         $OUT[836] = ($FLAG[330] OR NOT $FLAG[330] AND NOT $FLAG[331] AND NOT $FLAG[332]) AND NOT $FLAG[537]
      ;ENDFOLD
      ;FOLD A860 = (F330 + !F330 & !F331 & !F332) & F537 ;%{SE}%MKUKATPVW %CVW_SPS %VBOASG %P 2:A860 = (F330 + !F330 & !F331 & !F332) & F537, 3: BOASG
         $OUT[860] = ($FLAG[330] OR NOT $FLAG[330] AND NOT $FLAG[331] AND NOT $FLAG[332]) AND $FLAG[537]
      ;ENDFOLD
      ;FOLD Schritt 43 = A4039 ;%{SE}%MKUKATPVW %CVW_SPS %VST_CON %P 2:Schritt 43 = A4039, 3: ST_CON
         IF $OUT[4039] THEN
            PREVSTEP = $APP_INT[5]
            $APP_INT[5] = 43
         ENDIF
      ;ENDFOLD
   ;ENDFOLD
   ;FOLD SCHRITT 43 -- ROB EZ1/SP1/KE1 SZ4 -- ;%{P}%MKUKATPVW,%CSTEP,%VST_NR,%P 1:SCHRITT, 2:43, 3: ROB EZ1/SP1/KE1 SZ4
      ;FOLD ;%{H}
         Case 43
      ;ENDFOLD
      ;FOLD -- RSK Fehlerausgabe KF1/KW1 Initiator/Motor -- ;%{SE}%MKUKATPVW %CVW_COM %VCOMMENT %P 2:-- RSK Fehlerausgabe KF1/KW1 Initiator/Motor --, 3: VW_COMMENT
      ;ENDFOLD
      ;FOLD F322 = !F313 ;%{SE}%MKUKATPVW %CVW_SPS %VBOASG %P 2:F322 = !F313, 3: BOASG
         $FLAG[322] = NOT $FLAG[313]
      ;ENDFOLD
      ;FOLD T7 ( EIN ) = STOP ;%{SE}%MKUKATPVW %CVW_SPS %VTSTOP %P 2:T7 ( EIN ) = STOP, 3: TSTOP
         VW(#SET_TIME,TRUE,7,1,0)
      ;ENDFOLD
      ;FOLD A834 = !F322 & !F537 ;%{SE}%MKUKATPVW %CVW_SPS %VBOASG %P 2:A834 = !F322 & !F537, 3: BOASG
         $OUT[834] = NOT $FLAG[322] AND NOT $FLAG[537]
      ;ENDFOLD
      ;FOLD A858 = !F322 & F537 ;%{SE}%MKUKATPVW %CVW_SPS %VBOASG %P 2:A858 = !F322 & F537, 3: BOASG
         $OUT[858] = NOT $FLAG[322] AND $FLAG[537]
      ;ENDFOLD
      ;FOLD Schritt 44 = !F322 & A4039 ;%{SE}%MKUKATPVW %CVW_SPS %VST_CON %P 2:Schritt 44 = !F322 & A4039, 3: ST_CON
         IF NOT $FLAG[322] AND $OUT[4039] THEN
            PREVSTEP = $APP_INT[5]
            $APP_INT[5] = 44
         ENDIF
      ;ENDFOLD
      ;FOLD Schritt 46 = F322 & A4039 ;%{SE}%MKUKATPVW %CVW_SPS %VST_CON %P 2:Schritt 46 = F322 & A4039, 3: ST_CON
         IF $FLAG[322] AND $OUT[4039] THEN
            PREVSTEP = $APP_INT[5]
            $APP_INT[5] = 46
         ENDIF
      ;ENDFOLD
   ;ENDFOLD
   ;FOLD SCHRITT 44 -- ROB EZ1/SP1/KE1 SZ4 -- ;%{P}%MKUKATPVW,%CSTEP,%VST_NR,%P 1:SCHRITT, 2:44, 3: ROB EZ1/SP1/KE1 SZ4
      ;FOLD ;%{H}
         Case 44
      ;ENDFOLD
      ;FOLD F312 = AUS ;%{SE}%MKUKATPVW %CVW_SPS %VBOASG %P 2:F312 = AUS, 3: BOASG
         $FLAG[312] = FALSE
      ;ENDFOLD
      ;FOLD F313 = AUS ;%{SE}%MKUKATPVW %CVW_SPS %VBOASG %P 2:F313 = AUS, 3: BOASG
         $FLAG[313] = FALSE
      ;ENDFOLD
      ;FOLD -- Umdreh. KF setzen -- ;%{SE}%MKUKATPVW %CVW_COM %VCOMMENT %P 2:-- Umdreh. KF setzen --, 3: VW_COMMENT
      ;ENDFOLD
      ;FOLD i1 ( EIN ) = 0 ;%{SE}%MKUKATPVW %CVW_SPS %VARIASG %P 2:i1 ( EIN ) = 0, 3: ARIASG
         VW(#COUNTER,TRUE,1,0)
      ;ENDFOLD
      ;FOLD -- Ueberwachungszeit EZ1/SP1/KE1 SZ4 schliessen -- ;%{SE}%MKUKATPVW %CVW_COM %VCOMMENT %P 2:-- Ueberwachungszeit EZ1/SP1/KE1 SZ4 schliessen --, 3: VW_COMMENT
      ;ENDFOLD
      ;FOLD T9 ( EIN ) = -40[1/10Sek] ;%{SE}%MKUKATPVW %CVW_SPS %VTASG %P 2:T9 ( EIN ) = -40[1/10Sek], 3: TASG
         VW(#SET_TIME,TRUE,9,0,-40)
      ;ENDFOLD
      ;FOLD -- Ueberwachungszeit KF1 -- ;%{SE}%MKUKATPVW %CVW_COM %VCOMMENT %P 2:-- Ueberwachungszeit KF1 --, 3: VW_COMMENT
      ;ENDFOLD
      ;FOLD T7 ( EIN ) = -40[1/10Sek] ;%{SE}%MKUKATPVW %CVW_SPS %VTASG %P 2:T7 ( EIN ) = -40[1/10Sek], 3: TASG
         VW(#SET_TIME,TRUE,7,0,-40)
      ;ENDFOLD
      ;FOLD Schritt 45 = A4039 ;%{SE}%MKUKATPVW %CVW_SPS %VST_CON %P 2:Schritt 45 = A4039, 3: ST_CON
         IF $OUT[4039] THEN
            PREVSTEP = $APP_INT[5]
            $APP_INT[5] = 45
         ENDIF
      ;ENDFOLD
   ;ENDFOLD
   ;FOLD SCHRITT 45 -- ROB EZ1/SP1/KE1 SZ4 -- ;%{P}%MKUKATPVW,%CSTEP,%VST_NR,%P 1:SCHRITT, 2:45, 3: ROB EZ1/SP1/KE1 SZ4
      ;FOLD ;%{H}
         Case 45
      ;ENDFOLD
      ;FOLD -- KF1/KW1 Ausblasen -- ;%{SE}%MKUKATPVW %CVW_COM %VCOMMENT %P 2:-- KF1/KW1 Ausblasen --, 3: VW_COMMENT
      ;ENDFOLD
      ;FOLD A836 = (F330 + F331 + !F330 & !F331 & !F332) & !F537 ;%{SE}%MKUKATPVW %CVW_SPS %VBOASG %P 2:A836 = (F330 + F331 + !F330 & !F331 & !F332) & !F537, 3: BOASG
         $OUT[836] = ($FLAG[330] OR $FLAG[331] OR NOT $FLAG[330] AND NOT $FLAG[331] AND NOT $FLAG[332]) AND NOT $FLAG[537]
      ;ENDFOLD
      ;FOLD A860 = (F330 + F331 + !F330 & !F331 & !F332) & F537 ;%{SE}%MKUKATPVW %CVW_SPS %VBOASG %P 2:A860 = (F330 + F331 + !F330 & !F331 & !F332) & F537, 3: BOASG
         $OUT[860] = ($FLAG[330] OR $FLAG[331] OR NOT $FLAG[330] AND NOT $FLAG[331] AND NOT $FLAG[332]) AND $FLAG[537]
      ;ENDFOLD
      ;FOLD -- EZ1/SP1/KE1 SZ4 schliessen -- ;%{SE}%MKUKATPVW %CVW_COM %VCOMMENT %P 2:-- EZ1/SP1/KE1 SZ4 schliessen --, 3: VW_COMMENT
      ;ENDFOLD
      ;FOLD A717 = AUS ;%{SE}%MKUKATPVW %CVW_SPS %VBOASG %P 2:A717 = AUS, 3: BOASG
         $OUT[717] = FALSE
      ;ENDFOLD
      ;FOLD -- EZ1/SP1 -- ;%{SE}%MKUKATPVW %CVW_COM %VCOMMENT %P 2:-- EZ1/SP1 --, 3: VW_COMMENT
      ;ENDFOLD
      ;FOLD A718 = !F830 ;%{SE}%MKUKATPVW %CVW_SPS %VBOASG %P 2:A718 = !F830, 3: BOASG
         $OUT[718] = NOT $FLAG[830]
      ;ENDFOLD
      ;FOLD A766 = F830 ;%{SE}%MKUKATPVW %CVW_SPS %VBOASG %P 2:A766 = F830, 3: BOASG
         $OUT[766] = $FLAG[830]
      ;ENDFOLD
      ;FOLD Schritt 46 = (!E717 & E718 + T9) & A4039 ;%{SE}%MKUKATPVW %CVW_SPS %VST_CON %P 2:Schritt 46 = (!E717 & E718 + T9) & A4039, 3: ST_CON
         IF (NOT $IN[717] AND $IN[718] OR $TIMER_FLAG[9]) AND $OUT[4039] THEN
            PREVSTEP = $APP_INT[5]
            $APP_INT[5] = 46
         ENDIF
      ;ENDFOLD
   ;ENDFOLD
   ;FOLD SCHRITT 46 -- ROB EZ1/SP1/KE1 SZ4 -- ;%{P}%MKUKATPVW,%CSTEP,%VST_NR,%P 1:SCHRITT, 2:46, 3: ROB EZ1/SP1/KE1 SZ4
      ;FOLD ;%{H}
         Case 46
      ;ENDFOLD
      ;FOLD T9 ( EIN ) = STOP ;%{SE}%MKUKATPVW %CVW_SPS %VTSTOP %P 2:T9 ( EIN ) = STOP, 3: TSTOP
         VW(#SET_TIME,TRUE,9,1,0)
      ;ENDFOLD
      ;FOLD -- RSK Fehlerausgabe Kraftaufbau -- ;%{SE}%MKUKATPVW %CVW_COM %VCOMMENT %P 2:-- RSK Fehlerausgabe Kraftaufbau --, 3: VW_COMMENT
      ;ENDFOLD
      ;FOLD F325 = T9 ;%{SE}%MKUKATPVW %CVW_SPS %VBOASG %P 2:F325 = T9, 3: BOASG
         $FLAG[325] = $TIMER_FLAG[9]
      ;ENDFOLD
      ;FOLD -- KF1/KW1 abschalten bei Fehler -- ;%{SE}%MKUKATPVW %CVW_COM %VCOMMENT %P 2:-- KF1/KW1 abschalten bei Fehler --, 3: VW_COMMENT
      ;ENDFOLD
      ;FOLD A834 = !T7 & !T9 & !F537 ;%{SE}%MKUKATPVW %CVW_SPS %VBOASG %P 2:A834 = !T7 & !T9 & !F537, 3: BOASG
         $OUT[834] = NOT $TIMER_FLAG[7] AND NOT $TIMER_FLAG[9] AND NOT $FLAG[537]
      ;ENDFOLD
      ;FOLD A858 = !T7 & !T9 & F537 ;%{SE}%MKUKATPVW %CVW_SPS %VBOASG %P 2:A858 = !T7 & !T9 & F537, 3: BOASG
         $OUT[858] = NOT $TIMER_FLAG[7] AND NOT $TIMER_FLAG[9] AND $FLAG[537]
      ;ENDFOLD
      ;FOLD -- KF1/KW1 Ausblasen -- ;%{SE}%MKUKATPVW %CVW_COM %VCOMMENT %P 2:-- KF1/KW1 Ausblasen --, 3: VW_COMMENT
      ;ENDFOLD
      ;FOLD A836 = (F330 + F331 + !F330 & !F331 & !F332) & !T9 & !F537 ;%{SE}%MKUKATPVW %CVW_SPS %VBOASG %P 2:A836 = (F330 + F331 + !F330 & !F331 & !F332) & !T9 & !F537, 3: BOASG
         $OUT[836] = ($FLAG[330] OR $FLAG[331] OR NOT $FLAG[330] AND NOT $FLAG[331] AND NOT $FLAG[332]) AND NOT $TIMER_FLAG[9] AND NOT $FLAG[537]
      ;ENDFOLD
      ;FOLD A860 = (F330 + F331 + !F330 & !F331 & !F332) & !T9 & F537 ;%{SE}%MKUKATPVW %CVW_SPS %VBOASG %P 2:A860 = (F330 + F331 + !F330 & !F331 & !F332) & !T9 & F537, 3: BOASG
         $OUT[860] = ($FLAG[330] OR $FLAG[331] OR NOT $FLAG[330] AND NOT $FLAG[331] AND NOT $FLAG[332]) AND NOT $TIMER_FLAG[9] AND $FLAG[537]
      ;ENDFOLD
      ;FOLD -- Warte Fraesen fertig oder Timeout -- ;%{SE}%MKUKATPVW %CVW_COM %VCOMMENT %P 2:-- Warte Fraesen fertig oder Timeout --, 3: VW_COMMENT
      ;ENDFOLD
      ;FOLD Schritt 47 = (F116 & F79 + F112 & !F287 & F78 + F114 & F287 & F78 + T7 + T9) & A4039 ;%{SE}%MKUKATPVW %CVW_SPS %VST_CON %P 2:Schritt 47 = (F116 & F79 + F112 & !F287 & F78 + F114 & F287 & F78 + T7 + T9) & A4039, 3: ST_CON
         IF ($FLAG[116] AND $FLAG[79] OR $FLAG[112] AND NOT $FLAG[287] AND $FLAG[78] OR $FLAG[114] AND $FLAG[287] AND $FLAG[78] OR $TIMER_FLAG[7] OR $TIMER_FLAG[9]) AND $OUT[4039] THEN
            PREVSTEP = $APP_INT[5]
            $APP_INT[5] = 47
         ENDIF
      ;ENDFOLD
   ;ENDFOLD
   ;FOLD SCHRITT 47 -- ROB EZ1/SP1/KE1 SZ4 -- ;%{P}%MKUKATPVW,%CSTEP,%VST_NR,%P 1:SCHRITT, 2:47, 3: ROB EZ1/SP1/KE1 SZ4
      ;FOLD ;%{H}
         Case 47
      ;ENDFOLD
      ;FOLD -- Hilfsflag SK Programmwechsel -- ;%{SE}%MKUKATPVW %CVW_COM %VCOMMENT %P 2:-- Hilfsflag SK Programmwechsel --, 3: VW_COMMENT
      ;ENDFOLD
      ;FOLD F334 = AUS ;%{SE}%MKUKATPVW %CVW_SPS %VBOASG %P 2:F334 = AUS, 3: BOASG
         $FLAG[334] = FALSE
      ;ENDFOLD
      ;FOLD t7 ( EIN ) = STOP ;%{SE}%MKUKATPVW %CVW_SPS %VTSTOP %P 2:t7 ( EIN ) = STOP, 3: TSTOP
         VW(#SET_TIME,TRUE,7,1,0)
      ;ENDFOLD
      ;FOLD -- KF1/KW1 Ausblasen -- ;%{SE}%MKUKATPVW %CVW_COM %VCOMMENT %P 2:-- KF1/KW1 Ausblasen --, 3: VW_COMMENT
      ;ENDFOLD
      ;FOLD A836 = (F330 + F331 + F332 + !F330 & !F331 & !F332) & !F537 ;%{SE}%MKUKATPVW %CVW_SPS %VBOASG %P 2:A836 = (F330 + F331 + F332 + !F330 & !F331 & !F332) & !F537, 3: BOASG
         $OUT[836] = ($FLAG[330] OR $FLAG[331] OR $FLAG[332] OR NOT $FLAG[330] AND NOT $FLAG[331] AND NOT $FLAG[332]) AND NOT $FLAG[537]
      ;ENDFOLD
      ;FOLD A860 = (F330 + F331 + F332 + !F330 & !F331 & !F332) & F537 ;%{SE}%MKUKATPVW %CVW_SPS %VBOASG %P 2:A860 = (F330 + F331 + F332 + !F330 & !F331 & !F332) & F537, 3: BOASG
         $OUT[860] = ($FLAG[330] OR $FLAG[331] OR $FLAG[332] OR NOT $FLAG[330] AND NOT $FLAG[331] AND NOT $FLAG[332]) AND $FLAG[537]
      ;ENDFOLD
      ;FOLD -- KF Ausblasen Ausschaltverzoegerung starten -- ;%{SE}%MKUKATPVW %CVW_COM %VCOMMENT %P 2:-- KF Ausblasen Ausschaltverzoegerung starten --, 3: VW_COMMENT
      ;ENDFOLD
      ;FOLD F736 = EIN ;%{SE}%MKUKATPVW %CVW_SPS %VBOASG %P 2:F736 = EIN, 3: BOASG
         $FLAG[736] = TRUE
      ;ENDFOLD
      ;FOLD -- EZ1/SP1/KE1 SZ4 oeffnen -- ;%{SE}%MKUKATPVW %CVW_COM %VCOMMENT %P 2:-- EZ1/SP1/KE1 SZ4 oeffnen --, 3: VW_COMMENT
      ;ENDFOLD
      ;FOLD A718 = AUS ;%{SE}%MKUKATPVW %CVW_SPS %VBOASG %P 2:A718 = AUS, 3: BOASG
         $OUT[718] = FALSE
      ;ENDFOLD
      ;FOLD A766 = AUS ;%{SE}%MKUKATPVW %CVW_SPS %VBOASG %P 2:A766 = AUS, 3: BOASG
         $OUT[766] = FALSE
      ;ENDFOLD
      ;FOLD A717 = EIN ;%{SE}%MKUKATPVW %CVW_SPS %VBOASG %P 2:A717 = EIN, 3: BOASG
         $OUT[717] = TRUE
      ;ENDFOLD
      ;FOLD -- RSK Sammelstoerung -- ;%{SE}%MKUKATPVW %CVW_COM %VCOMMENT %P 2:-- RSK Sammelstoerung --, 3: VW_COMMENT
      ;ENDFOLD
      ;FOLD F329 = T7 + T9 ;%{SE}%MKUKATPVW %CVW_SPS %VBOASG %P 2:F329 = T7 + T9, 3: BOASG
         $FLAG[329] = $TIMER_FLAG[7] OR $TIMER_FLAG[9]
      ;ENDFOLD
      ;FOLD -- Hilfsflag Startfraesen -- ;%{SE}%MKUKATPVW %CVW_COM %VCOMMENT %P 2:-- Hilfsflag Startfraesen --, 3: VW_COMMENT
      ;ENDFOLD
      ;FOLD F114 = (F114 & F78 + F116 & F79) & F287 ;%{SE}%MKUKATPVW %CVW_SPS %VBOASG %P 2:F114 = (F114 & F78 + F116 & F79) & F287, 3: BOASG
         $FLAG[114] = ($FLAG[114] AND $FLAG[78] OR $FLAG[116] AND $FLAG[79]) AND $FLAG[287]
      ;ENDFOLD
      ;FOLD F116 = !F130 & F116 + F130 & F287 & F116 ;%{SE}%MKUKATPVW %CVW_SPS %VBOASG %P 2:F116 = !F130 & F116 + F130 & F287 & F116, 3: BOASG
         $FLAG[116] = NOT $FLAG[130] AND $FLAG[116] OR $FLAG[130] AND $FLAG[287] AND $FLAG[116]
      ;ENDFOLD
      ;FOLD F287 = F78 + F79 & F130 ;%{SE}%MKUKATPVW %CVW_SPS %VBOASG %P 2:F287 = F78 + F79 & F130, 3: BOASG
         $FLAG[287] = $FLAG[78] OR $FLAG[79] AND $FLAG[130]
      ;ENDFOLD
      ;FOLD -- Wiederholung beim Startfraesen -- ;%{SE}%MKUKATPVW %CVW_COM %VCOMMENT %P 2:-- Wiederholung beim Startfraesen --, 3: VW_COMMENT
      ;ENDFOLD
      ;FOLD Schritt 44 = E717 & !E718 & (F78 & !F114 + F79 & F130 & !F114) & !F329 & A4039 ;%{SE}%MKUKATPVW %CVW_SPS %VST_CON %P 2:Schritt 44 = E717 & !E718 & (F78 & !F114 + F79 & F130 & !F114) & !F329 & A4039, 3: ST_CON
         IF $IN[717] AND NOT $IN[718] AND ($FLAG[78] AND NOT $FLAG[114] OR $FLAG[79] AND $FLAG[130] AND NOT $FLAG[114]) AND NOT $FLAG[329] AND $OUT[4039] THEN
            PREVSTEP = $APP_INT[5]
            $APP_INT[5] = 44
         ENDIF
      ;ENDFOLD
      ;FOLD -- Weiter wenn Fraesen fertig -- ;%{SE}%MKUKATPVW %CVW_COM %VCOMMENT %P 2:-- Weiter wenn Fraesen fertig --, 3: VW_COMMENT
      ;ENDFOLD
      ;FOLD Schritt 48 = E717 & !E718 & (F79 & F116 & (!F130 + F114) + F78 & F114 + F329) & A4039 ;%{SE}%MKUKATPVW %CVW_SPS %VST_CON %P 2:Schritt 48 = E717 & !E718 & (F79 & F116 & (!F130 + F114) + F78 & F114 + F329) & A4039, 3: ST_CON
         IF $IN[717] AND NOT $IN[718] AND ($FLAG[79] AND $FLAG[116] AND (NOT $FLAG[130] OR $FLAG[114]) OR $FLAG[78] AND $FLAG[114] OR $FLAG[329]) AND $OUT[4039] THEN
            PREVSTEP = $APP_INT[5]
            $APP_INT[5] = 48
         ENDIF
      ;ENDFOLD
      ;FOLD -- Weiter bei Fehler -- ;%{SE}%MKUKATPVW %CVW_COM %VCOMMENT %P 2:-- Weiter bei Fehler --, 3: VW_COMMENT
      ;ENDFOLD
      ;FOLD Schritt 50 = F325 & (E26 + E27) & A4039 ;%{SE}%MKUKATPVW %CVW_SPS %VST_CON %P 2:Schritt 50 = F325 & (E26 + E27) & A4039, 3: ST_CON
         IF $FLAG[325] AND ($IN[26] OR $IN[27]) AND $OUT[4039] THEN
            PREVSTEP = $APP_INT[5]
            $APP_INT[5] = 50
         ENDIF
      ;ENDFOLD
   ;ENDFOLD
   ;FOLD SCHRITT 48 -- ROB EZ1/SP1/KE1 SZ4 -- ;%{P}%MKUKATPVW,%CSTEP,%VST_NR,%P 1:SCHRITT, 2:48, 3: ROB EZ1/SP1/KE1 SZ4
      ;FOLD ;%{H}
         Case 48
      ;ENDFOLD
      ;FOLD A717 = AUS ;%{SE}%MKUKATPVW %CVW_SPS %VBOASG %P 2:A717 = AUS, 3: BOASG
         $OUT[717] = FALSE
      ;ENDFOLD
      ;FOLD -- KF1/KW1 abschalten -- ;%{SE}%MKUKATPVW %CVW_COM %VCOMMENT %P 2:-- KF1/KW1 abschalten --, 3: VW_COMMENT
      ;ENDFOLD
      ;FOLD A834 = AUS ;%{SE}%MKUKATPVW %CVW_SPS %VBOASG %P 2:A834 = AUS, 3: BOASG
         $OUT[834] = FALSE
      ;ENDFOLD
      ;FOLD A858 = AUS ;%{SE}%MKUKATPVW %CVW_SPS %VBOASG %P 2:A858 = AUS, 3: BOASG
         $OUT[858] = FALSE
      ;ENDFOLD
      ;FOLD bin3 ( !F329 ) = 4 ;%{SE}%MKUKATPVW %CVW_SPS %VARIASG %P 2:bin3 ( !F329 ) = 4, 3: ARIASG
         VW(#BINOUT,NOT $FLAG[329],3,4)
      ;ENDFOLD
      ;FOLD -- Wartezeit Programmwechsel SK -- ;%{SE}%MKUKATPVW %CVW_COM %VCOMMENT %P 2:-- Wartezeit Programmwechsel SK --, 3: VW_COMMENT
      ;ENDFOLD
      ;FOLD T8 ( !F334 ) = -2[1/10Sek] ;%{SE}%MKUKATPVW %CVW_SPS %VTASG %P 2:T8 ( !F334 ) = -2[1/10Sek], 3: TASG
         VW(#SET_TIME,NOT $FLAG[334],8,0,-2)
      ;ENDFOLD
      ;FOLD -- Hilfsflag SK Programmwechsel -- ;%{SE}%MKUKATPVW %CVW_COM %VCOMMENT %P 2:-- Hilfsflag SK Programmwechsel --, 3: VW_COMMENT
      ;ENDFOLD
      ;FOLD F334 = EIN ;%{SE}%MKUKATPVW %CVW_SPS %VBOASG %P 2:F334 = EIN, 3: BOASG
         $FLAG[334] = TRUE
      ;ENDFOLD
      ;FOLD Schritt 49 = T8 & A4039 ;%{SE}%MKUKATPVW %CVW_SPS %VST_CON %P 2:Schritt 49 = T8 & A4039, 3: ST_CON
         IF $TIMER_FLAG[8] AND $OUT[4039] THEN
            PREVSTEP = $APP_INT[5]
            $APP_INT[5] = 49
         ENDIF
      ;ENDFOLD
   ;ENDFOLD
   ;FOLD SCHRITT 49 -- ROB EZ1/SP1/KE1 SZ4 -- ;%{P}%MKUKATPVW,%CSTEP,%VST_NR,%P 1:SCHRITT, 2:49, 3: ROB EZ1/SP1/KE1 SZ4
      ;FOLD ;%{H}
         Case 49
      ;ENDFOLD
      ;FOLD -- Hilfsflag SK Programmwechsel -- ;%{SE}%MKUKATPVW %CVW_COM %VCOMMENT %P 2:-- Hilfsflag SK Programmwechsel --, 3: VW_COMMENT
      ;ENDFOLD
      ;FOLD F334 = AUS ;%{SE}%MKUKATPVW %CVW_SPS %VBOASG %P 2:F334 = AUS, 3: BOASG
         $FLAG[334] = FALSE
      ;ENDFOLD
      ;FOLD -- Quitt. Fraesen SK1 -- ;%{SE}%MKUKATPVW %CVW_COM %VCOMMENT %P 2:-- Quitt. Fraesen SK1 --, 3: VW_COMMENT
      ;ENDFOLD
      ;FOLD A786 = !F329 & !F322 ;%{SE}%MKUKATPVW %CVW_SPS %VBOASG %P 2:A786 = !F329 & !F322, 3: BOASG
         $OUT[786] = NOT $FLAG[329] AND NOT $FLAG[322]
      ;ENDFOLD
      ;FOLD Schritt 50 = (!E786 & E787 & !E788 + F329) & A4039 ;%{SE}%MKUKATPVW %CVW_SPS %VST_CON %P 2:Schritt 50 = (!E786 & E787 & !E788 + F329) & A4039, 3: ST_CON
         IF (NOT $IN[786] AND $IN[787] AND NOT $IN[788] OR $FLAG[329]) AND $OUT[4039] THEN
            PREVSTEP = $APP_INT[5]
            $APP_INT[5] = 50
         ENDIF
      ;ENDFOLD
   ;ENDFOLD
   ;FOLD SCHRITT 50 -- ROB EZ1/SP1/KE1 SZ4 # Ende -- ;%{P}%MKUKATPVW,%CSTEP,%VST_NR,%P 1:SCHRITT, 2:50, 3: ROB EZ1/SP1/KE1 SZ4 # Ende
      ;FOLD ;%{H}
         Case 50
      ;ENDFOLD
      ;FOLD -- KF1/KW1 Ausblasen -- ;%{SE}%MKUKATPVW %CVW_COM %VCOMMENT %P 2:-- KF1/KW1 Ausblasen --, 3: VW_COMMENT
      ;ENDFOLD
      ;FOLD A836 = (F330 + F331 + F332) & F736 ;%{SE}%MKUKATPVW %CVW_SPS %VBOASG %P 2:A836 = (F330 + F331 + F332) & F736, 3: BOASG
         $OUT[836] = ($FLAG[330] OR $FLAG[331] OR $FLAG[332]) AND $FLAG[736]
      ;ENDFOLD
      ;FOLD A860 = (F330 + F331 + F332) & F736 ;%{SE}%MKUKATPVW %CVW_SPS %VBOASG %P 2:A860 = (F330 + F331 + F332) & F736, 3: BOASG
         $OUT[860] = ($FLAG[330] OR $FLAG[331] OR $FLAG[332]) AND $FLAG[736]
      ;ENDFOLD
      ;FOLD F91 = !E786 & E787 & !E788 & !F322 & !F325 & !F329 ;%{SE}%MKUKATPVW %CVW_SPS %VBOASG %P 2:F91 = !E786 & E787 & !E788 & !F322 & !F325 & !F329, 3: BOASG
         $FLAG[91] = NOT $IN[786] AND $IN[787] AND NOT $IN[788] AND NOT $FLAG[322] AND NOT $FLAG[325] AND NOT $FLAG[329]
      ;ENDFOLD
      ;FOLD Schritt 39 = (F322 + F325 + F329) & (E26 + E27) & A4039 ;%{SE}%MKUKATPVW %CVW_SPS %VST_CON %P 2:Schritt 39 = (F322 + F325 + F329) & (E26 + E27) & A4039, 3: ST_CON
         IF ($FLAG[322] OR $FLAG[325] OR $FLAG[329]) AND ($IN[26] OR $IN[27]) AND $OUT[4039] THEN
            PREVSTEP = $APP_INT[5]
            $APP_INT[5] = 39
         ENDIF
      ;ENDFOLD
      ;FOLD Schritt 1 = F91 & !F322 & !F325 & !F329 & A4039 ;%{SE}%MKUKATPVW %CVW_SPS %VST_CON %P 2:Schritt 1 = F91 & !F322 & !F325 & !F329 & A4039, 3: ST_CON
         IF $FLAG[91] AND NOT $FLAG[322] AND NOT $FLAG[325] AND NOT $FLAG[329] AND $OUT[4039] THEN
            PREVSTEP = $APP_INT[5]
            $APP_INT[5] = 1
         ENDIF
      ;ENDFOLD
   ;ENDFOLD
   ;FOLD SCHRITT 51 -- STAT EZ1/SP1/KE1 # Start-- ;%{P}%MKUKATPVW,%CSTEP,%VST_NR,%P 1:SCHRITT, 2:51, 3: STAT EZ1/SP1/KE1 # Start
      ;FOLD ;%{H}
         Case 51
      ;ENDFOLD
      ;FOLD -- RSK gestartet -- ;%{SE}%MKUKATPVW %CVW_COM %VCOMMENT %P 2:-- RSK gestartet --, 3: VW_COMMENT
      ;ENDFOLD
      ;FOLD F122 = AUS ;%{SE}%MKUKATPVW %CVW_SPS %VBOASG %P 2:F122 = AUS, 3: BOASG
         $FLAG[122] = FALSE
      ;ENDFOLD
      ;FOLD F321 = AUS ;%{SE}%MKUKATPVW %CVW_SPS %VBOASG %P 2:F321 = AUS, 3: BOASG
         $FLAG[321] = FALSE
      ;ENDFOLD
      ;FOLD F322 = AUS ;%{SE}%MKUKATPVW %CVW_SPS %VBOASG %P 2:F322 = AUS, 3: BOASG
         $FLAG[322] = FALSE
      ;ENDFOLD
      ;FOLD F323 = AUS ;%{SE}%MKUKATPVW %CVW_SPS %VBOASG %P 2:F323 = AUS, 3: BOASG
         $FLAG[323] = FALSE
      ;ENDFOLD
      ;FOLD F324 = AUS ;%{SE}%MKUKATPVW %CVW_SPS %VBOASG %P 2:F324 = AUS, 3: BOASG
         $FLAG[324] = FALSE
      ;ENDFOLD
      ;FOLD F325 = AUS ;%{SE}%MKUKATPVW %CVW_SPS %VBOASG %P 2:F325 = AUS, 3: BOASG
         $FLAG[325] = FALSE
      ;ENDFOLD
      ;FOLD F326 = AUS ;%{SE}%MKUKATPVW %CVW_SPS %VBOASG %P 2:F326 = AUS, 3: BOASG
         $FLAG[326] = FALSE
      ;ENDFOLD
      ;FOLD F327 = AUS ;%{SE}%MKUKATPVW %CVW_SPS %VBOASG %P 2:F327 = AUS, 3: BOASG
         $FLAG[327] = FALSE
      ;ENDFOLD
      ;FOLD F329 = AUS ;%{SE}%MKUKATPVW %CVW_SPS %VBOASG %P 2:F329 = AUS, 3: BOASG
         $FLAG[329] = FALSE
      ;ENDFOLD
      ;FOLD -- EZ1/SP1/KE1 SZ1 Zaehler -- ;%{SE}%MKUKATPVW %CVW_COM %VCOMMENT %P 2:-- EZ1/SP1/KE1 SZ1 Zaehler --, 3: VW_COMMENT
      ;ENDFOLD
      ;FOLD F94 = AUS ;%{SE}%MKUKATPVW %CVW_SPS %VBOASG %P 2:F94 = AUS, 3: BOASG
         $FLAG[94] = FALSE
      ;ENDFOLD
      ;FOLD F95 = AUS ;%{SE}%MKUKATPVW %CVW_SPS %VBOASG %P 2:F95 = AUS, 3: BOASG
         $FLAG[95] = FALSE
      ;ENDFOLD
      ;FOLD F96 = AUS ;%{SE}%MKUKATPVW %CVW_SPS %VBOASG %P 2:F96 = AUS, 3: BOASG
         $FLAG[96] = FALSE
      ;ENDFOLD
      ;FOLD F97 = AUS ;%{SE}%MKUKATPVW %CVW_SPS %VBOASG %P 2:F97 = AUS, 3: BOASG
         $FLAG[97] = FALSE
      ;ENDFOLD
      ;FOLD F98 = AUS ;%{SE}%MKUKATPVW %CVW_SPS %VBOASG %P 2:F98 = AUS, 3: BOASG
         $FLAG[98] = FALSE
      ;ENDFOLD
      ;FOLD F99 = AUS ;%{SE}%MKUKATPVW %CVW_SPS %VBOASG %P 2:F99 = AUS, 3: BOASG
         $FLAG[99] = FALSE
      ;ENDFOLD
      ;FOLD -- Hilfsflags Funktionstest KF Motor -- ;%{SE}%MKUKATPVW %CVW_COM %VCOMMENT %P 2:-- Hilfsflags Funktionstest KF Motor --, 3: VW_COMMENT
      ;ENDFOLD
      ;FOLD F312 = AUS ;%{SE}%MKUKATPVW %CVW_SPS %VBOASG %P 2:F312 = AUS, 3: BOASG
         $FLAG[312] = FALSE
      ;ENDFOLD
      ;FOLD F313 = AUS ;%{SE}%MKUKATPVW %CVW_SPS %VBOASG %P 2:F313 = AUS, 3: BOASG
         $FLAG[313] = FALSE
      ;ENDFOLD
      ;FOLD bin1 ( !F830 ) = 31 ;%{SE}%MKUKATPVW %CVW_SPS %VARIASG %P 2:bin1 ( !F830 ) = 31, 3: ARIASG
         VW(#BINOUT,NOT $FLAG[830],1,31)
      ;ENDFOLD
      ;FOLD bin3 ( EIN ) = 31 ;%{SE}%MKUKATPVW %CVW_SPS %VARIASG %P 2:bin3 ( EIN ) = 31, 3: ARIASG
         VW(#BINOUT,TRUE,3,31)
      ;ENDFOLD
      ;FOLD -- Wartezeit Programmwechsel SK -- ;%{SE}%MKUKATPVW %CVW_COM %VCOMMENT %P 2:-- Wartezeit Programmwechsel SK --, 3: VW_COMMENT
      ;ENDFOLD
      ;FOLD T8 ( !F334 ) = -2[1/10Sek] ;%{SE}%MKUKATPVW %CVW_SPS %VTASG %P 2:T8 ( !F334 ) = -2[1/10Sek], 3: TASG
         VW(#SET_TIME,NOT $FLAG[334],8,0,-2)
      ;ENDFOLD
      ;FOLD -- Hilfsflag SK Programmwechsel -- ;%{SE}%MKUKATPVW %CVW_COM %VCOMMENT %P 2:-- Hilfsflag SK Programmwechsel --, 3: VW_COMMENT
      ;ENDFOLD
      ;FOLD F334 = EIN ;%{SE}%MKUKATPVW %CVW_SPS %VBOASG %P 2:F334 = EIN, 3: BOASG
         $FLAG[334] = TRUE
      ;ENDFOLD
      ;FOLD -- Quitt. Fraesen SK1 AUS -- ;%{SE}%MKUKATPVW %CVW_COM %VCOMMENT %P 2:-- Quitt. Fraesen SK1 AUS --, 3: VW_COMMENT
      ;ENDFOLD
      ;FOLD A786 = AUS ;%{SE}%MKUKATPVW %CVW_SPS %VBOASG %P 2:A786 = AUS, 3: BOASG
         $OUT[786] = FALSE
      ;ENDFOLD
      ;FOLD Schritt 52 = T8 & A4039 ;%{SE}%MKUKATPVW %CVW_SPS %VST_CON %P 2:Schritt 52 = T8 & A4039, 3: ST_CON
         IF $TIMER_FLAG[8] AND $OUT[4039] THEN
            PREVSTEP = $APP_INT[5]
            $APP_INT[5] = 52
         ENDIF
      ;ENDFOLD
   ;ENDFOLD
   ;FOLD SCHRITT 52 -- STAT EZ1/SP1/KE1 -- ;%{P}%MKUKATPVW,%CSTEP,%VST_NR,%P 1:SCHRITT, 2:52, 3: STAT EZ1/SP1/KE1
      ;FOLD ;%{H}
         Case 52
      ;ENDFOLD
      ;FOLD -- Fraeszyklen fuer autom. KF-Umderhung -- ;%{SE}%MKUKATPVW %CVW_COM %VCOMMENT %P 2:-- Fraeszyklen fuer autom. KF-Umderhung --, 3: VW_COMMENT
      ;ENDFOLD
      ;FOLD i36 (EIN) = i36 + 1 ;%{SE}%MKUKATPVW %CVW_SPS %VARIASG %P 2:i36 (EIN) = i36 + 1, 3: ARIASG
         VW(#COUNTER,TRUE,36,$COUNT_I[36] + 1)
      ;ENDFOLD
      ;FOLD -- Hilfsflag SK Programmwechsel -- ;%{SE}%MKUKATPVW %CVW_COM %VCOMMENT %P 2:-- Hilfsflag SK Programmwechsel --, 3: VW_COMMENT
      ;ENDFOLD
      ;FOLD F334 = AUS ;%{SE}%MKUKATPVW %CVW_SPS %VBOASG %P 2:F334 = AUS, 3: BOASG
         $FLAG[334] = FALSE
      ;ENDFOLD
      ;FOLD -- Ueberwachungszeit KF1 EIN -- ;%{SE}%MKUKATPVW %CVW_COM %VCOMMENT %P 2:-- Ueberwachungszeit KF1 EIN --, 3: VW_COMMENT
      ;ENDFOLD
      ;FOLD T7 ( EIN ) = -50[1/10Sek] ;%{SE}%MKUKATPVW %CVW_SPS %VTASG %P 2:T7 ( EIN ) = -50[1/10Sek], 3: TASG
         VW(#SET_TIME,TRUE,7,0,-50)
      ;ENDFOLD
      ;FOLD -- KF1 einschalten -- ;%{SE}%MKUKATPVW %CVW_COM %VCOMMENT %P 2:-- KF1 einschalten --, 3: VW_COMMENT
      ;ENDFOLD
      ;FOLD i1 (EIN) = 0 ;%{SE}%MKUKATPVW %CVW_SPS %VARIASG %P 2:i1 (EIN) = 0, 3: ARIASG
         VW(#COUNTER,TRUE,1,0)
      ;ENDFOLD
      ;FOLD A834 = EIN ;%{SE}%MKUKATPVW %CVW_SPS %VBOASG %P 2:A834 = EIN, 3: BOASG
         $OUT[834] = TRUE
      ;ENDFOLD
      ;FOLD Schritt 53 = A4039 ;%{SE}%MKUKATPVW %CVW_SPS %VST_CON %P 2:Schritt 53 = A4039, 3: ST_CON
         IF $OUT[4039] THEN
            PREVSTEP = $APP_INT[5]
            $APP_INT[5] = 53
         ENDIF
      ;ENDFOLD
   ;ENDFOLD
   ;FOLD SCHRITT 53 -- STAT EZ1/SP1/KE1 -- ;%{P}%MKUKATPVW,%CSTEP,%VST_NR,%P 1:SCHRITT, 2:53, 3: STAT EZ1/SP1/KE1
      ;FOLD ;%{H}
         Case 53
      ;ENDFOLD
      ;FOLD -- Funktionstest KF Motor -- ;%{SE}%MKUKATPVW %CVW_COM %VCOMMENT %P 2:-- Funktionstest KF Motor --, 3: VW_COMMENT
      ;ENDFOLD
      ;FOLD F312 = EIN ;%{SE}%MKUKATPVW %CVW_SPS %VBOASG %P 2:F312 = EIN, 3: BOASG
         $FLAG[312] = TRUE
      ;ENDFOLD
      ;FOLD F313 = i1 > 2 ;%{SE}%MKUKATPVW %CVW_SPS %VBOCMP %P 2:F313 = i1 > 2, 3: BOCMP
         $FLAG[313] = $COUNT_I[1] > 2
      ;ENDFOLD
      ;FOLD Schritt 54 = (F313 + T7) & A4039 ;%{SE}%MKUKATPVW %CVW_SPS %VST_CON %P 2:Schritt 54 = (F313 + T7) & A4039, 3: ST_CON
         IF ($FLAG[313] OR $TIMER_FLAG[7]) AND $OUT[4039] THEN
            PREVSTEP = $APP_INT[5]
            $APP_INT[5] = 54
         ENDIF
      ;ENDFOLD
   ;ENDFOLD
   ;FOLD SCHRITT 54 -- STAT EZ1/SP1/KE1-- ;%{P}%MKUKATPVW,%CSTEP,%VST_NR,%P 1:SCHRITT, 2:54, 3: STAT EZ1/SP1/KE1
      ;FOLD ;%{H}
         Case 54
      ;ENDFOLD
      ;FOLD F312 = AUS ;%{SE}%MKUKATPVW %CVW_SPS %VBOASG %P 2:F312 = AUS, 3: BOASG
         $FLAG[312] = FALSE
      ;ENDFOLD
      ;FOLD -- Ueberwachungszeit KS1 schwenken -- ;%{SE}%MKUKATPVW %CVW_COM %VCOMMENT %P 2:-- Ueberwachungszeit KS1 schwenken --, 3: VW_COMMENT
      ;ENDFOLD
      ;FOLD t8 ( EIN ) = -100[1/10Sek] ;%{SE}%MKUKATPVW %CVW_SPS %VTASG %P 2:t8 ( EIN ) = -100[1/10Sek], 3: TASG
         VW(#SET_TIME,TRUE,8,0,-100)
      ;ENDFOLD
      ;FOLD Schritt 55 = A4039 ;%{SE}%MKUKATPVW %CVW_SPS %VST_CON %P 2:Schritt 55 = A4039, 3: ST_CON
         IF $OUT[4039] THEN
            PREVSTEP = $APP_INT[5]
            $APP_INT[5] = 55
         ENDIF
      ;ENDFOLD
   ;ENDFOLD
   ;FOLD SCHRITT 55 -- STAT EZ1/SP1/KE1 -- ;%{P}%MKUKATPVW,%CSTEP,%VST_NR,%P 1:SCHRITT, 2:55, 3: STAT EZ1/SP1/KE1
      ;FOLD ;%{H}
         Case 55
      ;ENDFOLD
      ;FOLD -- RSK Fehlerausgabe KF1 Initiator/Motor -- ;%{SE}%MKUKATPVW %CVW_COM %VCOMMENT %P 2:-- RSK Fehlerausgabe KF1 Initiator/Motor --, 3: VW_COMMENT
      ;ENDFOLD
      ;FOLD F322 = !F313 ;%{SE}%MKUKATPVW %CVW_SPS %VBOASG %P 2:F322 = !F313, 3: BOASG
         $FLAG[322] = NOT $FLAG[313]
      ;ENDFOLD
      ;FOLD -- RSK Fehlerausgabe KS1 Ruhest. -- ;%{SE}%MKUKATPVW %CVW_COM %VCOMMENT %P 2:-- RSK Fehlerausgabe KS1 Ruhest. --, 3: VW_COMMENT
      ;ENDFOLD
      ;FOLD F323 = (!E836 + E837 + E838 + !E839) & !F324 & !F328 ;%{SE}%MKUKATPVW %CVW_SPS %VBOASG %P 2:F323 = (!E836 + E837 + E838 + !E839) & !F324 & !F328, 3: BOASG
         $FLAG[323] = (NOT $IN[836] OR $IN[837] OR $IN[838] OR NOT $IN[839]) AND NOT $FLAG[324] AND NOT $FLAG[328]
      ;ENDFOLD
      ;FOLD -- RSK Sammelstoerung -- ;%{SE}%MKUKATPVW %CVW_COM %VCOMMENT %P 2:-- RSK Sammelstoerung --, 3: VW_COMMENT
      ;ENDFOLD
      ;FOLD F329 = F322 + F323 + T8 ;%{SE}%MKUKATPVW %CVW_SPS %VBOASG %P 2:F329 = F322 + F323 + T8, 3: BOASG
         $FLAG[329] = $FLAG[322] OR $FLAG[323] OR $TIMER_FLAG[8]
      ;ENDFOLD
      ;FOLD T7 ( EIN ) = STOP ;%{SE}%MKUKATPVW %CVW_SPS %VTSTOP %P 2:T7 ( EIN ) = STOP, 3: TSTOP
         VW(#SET_TIME,TRUE,7,1,0)
      ;ENDFOLD
      ;FOLD A834 = !F322 & !F323 ;%{SE}%MKUKATPVW %CVW_SPS %VBOASG %P 2:A834 = !F322 & !F323, 3: BOASG
         $OUT[834] = NOT $FLAG[322] AND NOT $FLAG[323]
      ;ENDFOLD
      ;FOLD -- KF1 Versetzeinheit vor -- ;%{SE}%MKUKATPVW %CVW_COM %VCOMMENT %P 2:-- KF1 Versetzeinheit vor --, 3: VW_COMMENT
      ;ENDFOLD
      ;FOLD A835 = !F322 & !F323 & F564 ;%{SE}%MKUKATPVW %CVW_SPS %VBOASG %P 2:A835 = !F322 & !F323 & F564, 3: BOASG
         $OUT[835] = NOT $FLAG[322] AND NOT $FLAG[323] AND $FLAG[564]
      ;ENDFOLD
      ;FOLD Schritt 56 = (!F322 & !F323 & (E835 & F564 + !E835 & !F564) + T8) & A4039 ;%{SE}%MKUKATPVW %CVW_SPS %VST_CON %P 2:Schritt 56 = (!F322 & !F323 & (E835 & F564 + !E835 & !F564) + T8) & A4039, 3: ST_CON
         IF (NOT $FLAG[322] AND NOT $FLAG[323] AND ($IN[835] AND $FLAG[564] OR NOT $IN[835] AND NOT $FLAG[564]) OR $TIMER_FLAG[8]) AND $OUT[4039] THEN
            PREVSTEP = $APP_INT[5]
            $APP_INT[5] = 56
         ENDIF
      ;ENDFOLD
      ;FOLD Schritt 72 = (F322 + F323) & !F324 & !F328 & A4039 ;%{SE}%MKUKATPVW %CVW_SPS %VST_CON %P 2:Schritt 72 = (F322 + F323) & !F324 & !F328 & A4039, 3: ST_CON
         IF ($FLAG[322] OR $FLAG[323]) AND NOT $FLAG[324] AND NOT $FLAG[328] AND $OUT[4039] THEN
            PREVSTEP = $APP_INT[5]
            $APP_INT[5] = 72
         ENDIF
      ;ENDFOLD
   ;ENDFOLD
   ;FOLD SCHRITT 56 -- STAT EZ1/SP1/KE1 -- ;%{P}%MKUKATPVW,%CSTEP,%VST_NR,%P 1:SCHRITT, 2:56, 3: STAT EZ1/SP1/KE1
      ;FOLD ;%{H}
         Case 56
      ;ENDFOLD
      ;FOLD -- RSK Sammelstoerung -- ;%{SE}%MKUKATPVW %CVW_COM %VCOMMENT %P 2:-- RSK Sammelstoerung --, 3: VW_COMMENT
      ;ENDFOLD
      ;FOLD F329 = T8 ;%{SE}%MKUKATPVW %CVW_SPS %VBOASG %P 2:F329 = T8, 3: BOASG
         $FLAG[329] = $TIMER_FLAG[8]
      ;ENDFOLD
      ;FOLD F324 = AUS ;%{SE}%MKUKATPVW %CVW_SPS %VBOASG %P 2:F324 = AUS, 3: BOASG
         $FLAG[324] = FALSE
      ;ENDFOLD
      ;FOLD F328 = AUS ;%{SE}%MKUKATPVW %CVW_SPS %VBOASG %P 2:F328 = AUS, 3: BOASG
         $FLAG[328] = FALSE
      ;ENDFOLD
      ;FOLD -- KS1 in Arbeitsstellung schwenken -- ;%{SE}%MKUKATPVW %CVW_COM %VCOMMENT %P 2:-- KS1 in Arbeitsstellung schwenken --, 3: VW_COMMENT
      ;ENDFOLD
      ;FOLD A840 = (F745 + !F714) & E717 & !E837 & (E835 & F564 + !E835 & !F564) ;%{SE}%MKUKATPVW %CVW_SPS %VBOASG %P 2:A840 = (F745 + !F714) & E717 & !E837 & (E835 & F564 + !E835 & !F564), 3: BOASG
         $OUT[840] = ($FLAG[745] OR NOT $FLAG[714]) AND $IN[717] AND NOT $IN[837] AND ($IN[835] AND $FLAG[564] OR NOT $IN[835] AND NOT $FLAG[564])
      ;ENDFOLD
      ;FOLD -- KF1 Ausblasen -- ;%{SE}%MKUKATPVW %CVW_COM %VCOMMENT %P 2:-- KF1 Ausblasen --, 3: VW_COMMENT
      ;ENDFOLD
      ;FOLD A836 = F330 + !F330 & !F331 & !F332 ;%{SE}%MKUKATPVW %CVW_SPS %VBOASG %P 2:A836 = F330 + !F330 & !F331 & !F332, 3: BOASG
         $OUT[836] = $FLAG[330] OR NOT $FLAG[330] AND NOT $FLAG[331] AND NOT $FLAG[332]
      ;ENDFOLD
      ;FOLD Schritt 57 = (F745 + !F714) & E717 & (A840 + E837 + T8) & A4039 ;%{SE}%MKUKATPVW %CVW_SPS %VST_CON %P 2:Schritt 57 = (F745 + !F714) & E717 & (A840 + E837 + T8) & A4039, 3: ST_CON
         IF ($FLAG[745] OR NOT $FLAG[714]) AND $IN[717] AND ($OUT[840] OR $IN[837] OR $TIMER_FLAG[8]) AND $OUT[4039] THEN
            PREVSTEP = $APP_INT[5]
            $APP_INT[5] = 57
         ENDIF
      ;ENDFOLD
   ;ENDFOLD
   ;FOLD SCHRITT 57 -- STAT EZ1/SP1/KE1 -- ;%{P}%MKUKATPVW,%CSTEP,%VST_NR,%P 1:SCHRITT, 2:57, 3: STAT EZ1/SP1/KE1
      ;FOLD ;%{H}
         Case 57
      ;ENDFOLD
      ;FOLD -- RSK Fehlerausgabe KF Versetzeinheit -- ;%{SE}%MKUKATPVW %CVW_COM %VCOMMENT %P 2:-- RSK Fehlerausgabe KF Versetzeinheit --, 3: VW_COMMENT
      ;ENDFOLD
      ;FOLD F328 = !E835 & F564 & !F324 ;%{SE}%MKUKATPVW %CVW_SPS %VBOASG %P 2:F328 = !E835 & F564 & !F324, 3: BOASG
         $FLAG[328] = NOT $IN[835] AND $FLAG[564] AND NOT $FLAG[324]
      ;ENDFOLD
      ;FOLD -- RSK Fehlerausgabe KS1 Arbeitsstellung -- ;%{SE}%MKUKATPVW %CVW_COM %VCOMMENT %P 2:-- RSK Fehlerausgabe KS1 Arbeitsstellung --, 3: VW_COMMENT
      ;ENDFOLD
      ;FOLD F324 = (E836 + !E837 + !E838 + E839) & T8 & (E835 + !F564) + F324 ;%{SE}%MKUKATPVW %CVW_SPS %VBOASG %P 2:F324 = (E836 + !E837 + !E838 + E839) & T8 & (E835 + !F564) + F324, 3: BOASG
         $FLAG[324] = ($IN[836] OR NOT $IN[837] OR NOT $IN[838] OR $IN[839]) AND $TIMER_FLAG[8] AND ($IN[835] OR NOT $FLAG[564]) OR $FLAG[324]
      ;ENDFOLD
      ;FOLD -- RSK Fehlerausgabe EZ/SP min. Oeffnung -- ;%{SE}%MKUKATPVW %CVW_COM %VCOMMENT %P 2:-- RSK Fehlerausgabe EZ/SP min. Oeffnung --, 3: VW_COMMENT
      ;ENDFOLD
      ;FOLD F333 = !F745 ;%{SE}%MKUKATPVW %CVW_SPS %VBOASG %P 2:F333 = !F745, 3: BOASG
         $FLAG[333] = NOT $FLAG[745]
      ;ENDFOLD
      ;FOLD -- RSK Sammelstoerung -- ;%{SE}%MKUKATPVW %CVW_COM %VCOMMENT %P 2:-- RSK Sammelstoerung --, 3: VW_COMMENT
      ;ENDFOLD
      ;FOLD F329 = F324 + F328 + F333 ;%{SE}%MKUKATPVW %CVW_SPS %VBOASG %P 2:F329 = F324 + F328 + F333, 3: BOASG
         $FLAG[329] = $FLAG[324] OR $FLAG[328] OR $FLAG[333]
      ;ENDFOLD
      ;FOLD A834 = !F324 & !F328 ;%{SE}%MKUKATPVW %CVW_SPS %VBOASG %P 2:A834 = !F324 & !F328, 3: BOASG
         $OUT[834] = NOT $FLAG[324] AND NOT $FLAG[328]
      ;ENDFOLD
      ;FOLD -- KF1 Ausblasen -- ;%{SE}%MKUKATPVW %CVW_COM %VCOMMENT %P 2:-- KF1 Ausblasen --, 3: VW_COMMENT
      ;ENDFOLD
      ;FOLD A836 = (F330 + !F330 & !F331 & !F332) & !F324 & !F328 ;%{SE}%MKUKATPVW %CVW_SPS %VBOASG %P 2:A836 = (F330 + !F330 & !F331 & !F332) & !F324 & !F328, 3: BOASG
         $OUT[836] = ($FLAG[330] OR NOT $FLAG[330] AND NOT $FLAG[331] AND NOT $FLAG[332]) AND NOT $FLAG[324] AND NOT $FLAG[328]
      ;ENDFOLD
      ;FOLD A836 = F564 ;%{SE}%MKUKATPVW %CVW_SPS %VBOASG %P 2:A836 = F564, 3: BOASG
         $OUT[836] = $FLAG[564]
      ;ENDFOLD
      ;FOLD -- Ueberwachungszeit EZ1/SP1/KE1 SZ1 schliessen -- ;%{SE}%MKUKATPVW %CVW_COM %VCOMMENT %P 2:-- Ueberwachungszeit EZ1/SP1/KE1 SZ1 schliessen --, 3: VW_COMMENT
      ;ENDFOLD
      ;FOLD t9 ( EIN ) = -80[1/10Sek] ;%{SE}%MKUKATPVW %CVW_SPS %VTASG %P 2:t9 ( EIN ) = -80[1/10Sek], 3: TASG
         VW(#SET_TIME,TRUE,9,0,-80)
      ;ENDFOLD
      ;FOLD -- Verweilzeit Versetzeinheit Rueck -- ;%{SE}%MKUKATPVW %CVW_COM %VCOMMENT %P 2:-- Verweilzeit Versetzeinheit Rueck --, 3: VW_COMMENT
      ;ENDFOLD
      ;FOLD t11 ( EIN ) = i24[1/10Sek] ;%{SE}%MKUKATPVW %CVW_SPS %VTASG %P 2:t11 ( EIN ) = i24[1/10Sek], 3: TASG
         VW(#SET_TIME,TRUE,11,0,$COUNT_I[24])
      ;ENDFOLD
      ;FOLD Schritt 52 = (F324 + F328) & (E26 + E27) & A4039 ;%{SE}%MKUKATPVW %CVW_SPS %VST_CON %P 2:Schritt 52 = (F324 + F328) & (E26 + E27) & A4039, 3: ST_CON
         IF ($FLAG[324] OR $FLAG[328]) AND ($IN[26] OR $IN[27]) AND $OUT[4039] THEN
            PREVSTEP = $APP_INT[5]
            $APP_INT[5] = 52
         ENDIF
      ;ENDFOLD
      ;FOLD Schritt 58 = !F324 & !F328 & !E836 & E837 & E838 & !E839 & A4039 ;%{SE}%MKUKATPVW %CVW_SPS %VST_CON %P 2:Schritt 58 = !F324 & !F328 & !E836 & E837 & E838 & !E839 & A4039, 3: ST_CON
         IF NOT $FLAG[324] AND NOT $FLAG[328] AND NOT $IN[836] AND $IN[837] AND $IN[838] AND NOT $IN[839] AND $OUT[4039] THEN
            PREVSTEP = $APP_INT[5]
            $APP_INT[5] = 58
         ENDIF
      ;ENDFOLD
   ;ENDFOLD
   ;FOLD SCHRITT 58 -- STAT EZ1/SP1/KE1-- ;%{P}%MKUKATPVW,%CSTEP,%VST_NR,%P 1:SCHRITT, 2:58, 3: STAT EZ1/SP1/KE1
      ;FOLD ;%{H}
         Case 58
      ;ENDFOLD
      ;FOLD -- Umdreh. KF setzen zwischenspeichern -- ;%{SE}%MKUKATPVW %CVW_COM %VCOMMENT %P 2:-- Umdreh. KF setzen zwischenspeichern --, 3: VW_COMMENT
      ;ENDFOLD
      ;FOLD i45 ( EIN ) = i4 ;%{SE}%MKUKATPVW %CVW_SPS %VARIASG %P 2:i45 ( EIN ) = i4, 3: ARIASG
         VW(#COUNTER,TRUE,45,$COUNT_I[4])
      ;ENDFOLD
      ;FOLD i4 ( F99 ) = i33 ;%{SE}%MKUKATPVW %CVW_SPS %VARIASG %P 2:i4 ( F99 ) = i33, 3: ARIASG
         VW(#COUNTER,$FLAG[99],4,$COUNT_I[33])
      ;ENDFOLD
      ;FOLD i1 ( EIN ) = 0 ;%{SE}%MKUKATPVW %CVW_SPS %VARIASG %P 2:i1 ( EIN ) = 0, 3: ARIASG
         VW(#COUNTER,TRUE,1,0)
      ;ENDFOLD
      ;FOLD F98 = AUS ;%{SE}%MKUKATPVW %CVW_SPS %VBOASG %P 2:F98 = AUS, 3: BOASG
         $FLAG[98] = FALSE
      ;ENDFOLD
      ;FOLD F312 = AUS ;%{SE}%MKUKATPVW %CVW_SPS %VBOASG %P 2:F312 = AUS, 3: BOASG
         $FLAG[312] = FALSE
      ;ENDFOLD
      ;FOLD F313 = AUS ;%{SE}%MKUKATPVW %CVW_SPS %VBOASG %P 2:F313 = AUS, 3: BOASG
         $FLAG[313] = FALSE
      ;ENDFOLD
      ;FOLD F324 = AUS ;%{SE}%MKUKATPVW %CVW_SPS %VBOASG %P 2:F324 = AUS, 3: BOASG
         $FLAG[324] = FALSE
      ;ENDFOLD
      ;FOLD F328 = AUS ;%{SE}%MKUKATPVW %CVW_SPS %VBOASG %P 2:F328 = AUS, 3: BOASG
         $FLAG[328] = FALSE
      ;ENDFOLD
      ;FOLD -- KF1 einschalten nach Fehler -- ;%{SE}%MKUKATPVW %CVW_COM %VCOMMENT %P 2:-- KF1 einschalten nach Fehler --, 3: VW_COMMENT
      ;ENDFOLD
      ;FOLD A834 = EIN ;%{SE}%MKUKATPVW %CVW_SPS %VBOASG %P 2:A834 = EIN, 3: BOASG
         $OUT[834] = TRUE
      ;ENDFOLD
      ;FOLD -- KF1 Versetzeinheit rueck -- ;%{SE}%MKUKATPVW %CVW_COM %VCOMMENT %P 2:-- KF1 Versetzeinheit rueck --, 3: VW_COMMENT
      ;ENDFOLD
      ;FOLD A835 = AUS ;%{SE}%MKUKATPVW %CVW_SPS %VBOASG %P 2:A835 = AUS, 3: BOASG
         $OUT[835] = FALSE
      ;ENDFOLD
      ;FOLD Schritt 59 = T11 & A4039 ;%{SE}%MKUKATPVW %CVW_SPS %VST_CON %P 2:Schritt 59 = T11 & A4039, 3: ST_CON
         IF $TIMER_FLAG[11] AND $OUT[4039] THEN
            PREVSTEP = $APP_INT[5]
            $APP_INT[5] = 59
         ENDIF
      ;ENDFOLD
   ;ENDFOLD
   ;FOLD SCHRITT 59 -- STAT EZ1/SP1/KE1 -- ;%{P}%MKUKATPVW,%CSTEP,%VST_NR,%P 1:SCHRITT, 2:59, 3: STAT EZ1/SP1/KE1
      ;FOLD ;%{H}
         Case 59
      ;ENDFOLD
      ;FOLD t11 ( EIN ) = STOP ;%{SE}%MKUKATPVW %CVW_SPS %VTSTOP %P 2:t11 ( EIN ) = STOP, 3: TSTOP
         VW(#SET_TIME,TRUE,11,1,0)
      ;ENDFOLD
      ;FOLD -- EZ1/SP1/KE1 SZ1 schliessen -- ;%{SE}%MKUKATPVW %CVW_COM %VCOMMENT %P 2:-- EZ1/SP1/KE1 SZ1 schliessen --, 3: VW_COMMENT
      ;ENDFOLD
      ;FOLD A717 = AUS ;%{SE}%MKUKATPVW %CVW_SPS %VBOASG %P 2:A717 = AUS, 3: BOASG
         $OUT[717] = FALSE
      ;ENDFOLD
      ;FOLD -- EZ1/SP1 -- ;%{SE}%MKUKATPVW %CVW_COM %VCOMMENT %P 2:-- EZ1/SP1 --, 3: VW_COMMENT
      ;ENDFOLD
      ;FOLD A718 = !F830 ;%{SE}%MKUKATPVW %CVW_SPS %VBOASG %P 2:A718 = !F830, 3: BOASG
         $OUT[718] = NOT $FLAG[830]
      ;ENDFOLD
      ;FOLD A766 = F830 ;%{SE}%MKUKATPVW %CVW_SPS %VBOASG %P 2:A766 = F830, 3: BOASG
         $OUT[766] = $FLAG[830]
      ;ENDFOLD
      ;FOLD -- KF1 Ausblasen -- ;%{SE}%MKUKATPVW %CVW_COM %VCOMMENT %P 2:-- KF1 Ausblasen --, 3: VW_COMMENT
      ;ENDFOLD
      ;FOLD A836 = F330 + F331 + !F330 & !F331 & !F332 ;%{SE}%MKUKATPVW %CVW_SPS %VBOASG %P 2:A836 = F330 + F331 + !F330 & !F331 & !F332, 3: BOASG
         $OUT[836] = $FLAG[330] OR $FLAG[331] OR NOT $FLAG[330] AND NOT $FLAG[331] AND NOT $FLAG[332]
      ;ENDFOLD
      ;FOLD Schritt 60 = (!E717 & E718 + T9) & A4039 ;%{SE}%MKUKATPVW %CVW_SPS %VST_CON %P 2:Schritt 60 = (!E717 & E718 + T9) & A4039, 3: ST_CON
         IF (NOT $IN[717] AND $IN[718] OR $TIMER_FLAG[9]) AND $OUT[4039] THEN
            PREVSTEP = $APP_INT[5]
            $APP_INT[5] = 60
         ENDIF
      ;ENDFOLD
   ;ENDFOLD
   ;FOLD SCHRITT 60 -- STAT EZ1/SP1/KE1 -- ;%{P}%MKUKATPVW,%CSTEP,%VST_NR,%P 1:SCHRITT, 2:60, 3: STAT EZ1/SP1/KE1
      ;FOLD ;%{H}
         Case 60
      ;ENDFOLD
      ;FOLD -- RSK Fehlerausgabe Kraftaufbau -- ;%{SE}%MKUKATPVW %CVW_COM %VCOMMENT %P 2:-- RSK Fehlerausgabe Kraftaufbau --, 3: VW_COMMENT
      ;ENDFOLD
      ;FOLD F325 = T9 ;%{SE}%MKUKATPVW %CVW_SPS %VBOASG %P 2:F325 = T9, 3: BOASG
         $FLAG[325] = $TIMER_FLAG[9]
      ;ENDFOLD
      ;FOLD -- RSK Sammelstoerung -- ;%{SE}%MKUKATPVW %CVW_COM %VCOMMENT %P 2:-- RSK Sammelstoerung --, 3: VW_COMMENT
      ;ENDFOLD
      ;FOLD F329 = F325 ;%{SE}%MKUKATPVW %CVW_SPS %VBOASG %P 2:F329 = F325, 3: BOASG
         $FLAG[329] = $FLAG[325]
      ;ENDFOLD
      ;FOLD -- KF1 abschalten bei Fehler -- ;%{SE}%MKUKATPVW %CVW_COM %VCOMMENT %P 2:-- KF1 abschalten bei Fehler --, 3: VW_COMMENT
      ;ENDFOLD
      ;FOLD A834 = !T9 ;%{SE}%MKUKATPVW %CVW_SPS %VBOASG %P 2:A834 = !T9, 3: BOASG
         $OUT[834] = NOT $TIMER_FLAG[9]
      ;ENDFOLD
      ;FOLD -- KF1 Ausblasen -- ;%{SE}%MKUKATPVW %CVW_COM %VCOMMENT %P 2:-- KF1 Ausblasen --, 3: VW_COMMENT
      ;ENDFOLD
      ;FOLD A836 = (F330 + F331 + !F330 & !F331 & !F332) & !T9 ;%{SE}%MKUKATPVW %CVW_SPS %VBOASG %P 2:A836 = (F330 + F331 + !F330 & !F331 & !F332) & !T9, 3: BOASG
         $OUT[836] = ($FLAG[330] OR $FLAG[331] OR NOT $FLAG[330] AND NOT $FLAG[331] AND NOT $FLAG[332]) AND NOT $TIMER_FLAG[9]
      ;ENDFOLD
      ;FOLD -- Warte Fraesen fertig oder Timeout -- ;%{SE}%MKUKATPVW %CVW_COM %VCOMMENT %P 2:-- Warte Fraesen fertig oder Timeout --, 3: VW_COMMENT
      ;ENDFOLD
      ;FOLD Schritt 61 = (F79 & F98 + F78 & F94 & !F287 + T7 + T9 + F325) & A4039 ;%{SE}%MKUKATPVW %CVW_SPS %VST_CON %P 2:Schritt 61 = (F79 & F98 + F78 & F94 & !F287 + T7 + T9 + F325) & A4039, 3: ST_CON
         IF ($FLAG[79] AND $FLAG[98] OR $FLAG[78] AND $FLAG[94] AND NOT $FLAG[287] OR $TIMER_FLAG[7] OR $TIMER_FLAG[9] OR $FLAG[325]) AND $OUT[4039] THEN
            PREVSTEP = $APP_INT[5]
            $APP_INT[5] = 61
         ENDIF
      ;ENDFOLD
      ;FOLD Schritt 61 = (F78 & F96 & F287 + T7 + T9 + F325) & A4039 ;%{SE}%MKUKATPVW %CVW_SPS %VST_CON %P 2:Schritt 61 = (F78 & F96 & F287 + T7 + T9 + F325) & A4039, 3: ST_CON
         IF ($FLAG[78] AND $FLAG[96] AND $FLAG[287] OR $TIMER_FLAG[7] OR $TIMER_FLAG[9] OR $FLAG[325]) AND $OUT[4039] THEN
            PREVSTEP = $APP_INT[5]
            $APP_INT[5] = 61
         ENDIF
      ;ENDFOLD
   ;ENDFOLD
   ;FOLD SCHRITT 61 -- STAT EZ1/SP1/KE1-- ;%{P}%MKUKATPVW,%CSTEP,%VST_NR,%P 1:SCHRITT, 2:61, 3: STAT EZ1/SP1/KE1
      ;FOLD ;%{H}
         Case 61
      ;ENDFOLD
      ;FOLD -- EZ1/SP1/KE1 SZ1 oeffnen -- ;%{SE}%MKUKATPVW %CVW_COM %VCOMMENT %P 2:-- EZ1/SP1/KE1 SZ1 oeffnen --, 3: VW_COMMENT
      ;ENDFOLD
      ;FOLD t9 ( EIN ) = STOP ;%{SE}%MKUKATPVW %CVW_SPS %VTSTOP %P 2:t9 ( EIN ) = STOP, 3: TSTOP
         VW(#SET_TIME,TRUE,9,1,0)
      ;ENDFOLD
      ;FOLD A718 = AUS ;%{SE}%MKUKATPVW %CVW_SPS %VBOASG %P 2:A718 = AUS, 3: BOASG
         $OUT[718] = FALSE
      ;ENDFOLD
      ;FOLD A766 = AUS ;%{SE}%MKUKATPVW %CVW_SPS %VBOASG %P 2:A766 = AUS, 3: BOASG
         $OUT[766] = FALSE
      ;ENDFOLD
      ;FOLD A717 = EIN ;%{SE}%MKUKATPVW %CVW_SPS %VBOASG %P 2:A717 = EIN, 3: BOASG
         $OUT[717] = TRUE
      ;ENDFOLD
      ;FOLD -- KF1 Ausblasen -- ;%{SE}%MKUKATPVW %CVW_COM %VCOMMENT %P 2:-- KF1 Ausblasen --, 3: VW_COMMENT
      ;ENDFOLD
      ;FOLD A836 = (F330 + F331 + F332 + !F330 & !F331 & !F332) & !T9 ;%{SE}%MKUKATPVW %CVW_SPS %VBOASG %P 2:A836 = (F330 + F331 + F332 + !F330 & !F331 & !F332) & !T9, 3: BOASG
         $OUT[836] = ($FLAG[330] OR $FLAG[331] OR $FLAG[332] OR NOT $FLAG[330] AND NOT $FLAG[331] AND NOT $FLAG[332]) AND NOT $TIMER_FLAG[9]
      ;ENDFOLD
      ;FOLD -- KF Ausblasen Ausschaltverzoegerung starten -- ;%{SE}%MKUKATPVW %CVW_COM %VCOMMENT %P 2:-- KF Ausblasen Ausschaltverzoegerung starten --, 3: VW_COMMENT
      ;ENDFOLD
      ;FOLD F737 = EIN ;%{SE}%MKUKATPVW %CVW_SPS %VBOASG %P 2:F737 = EIN, 3: BOASG
         $FLAG[737] = TRUE
      ;ENDFOLD
      ;FOLD -- RSK Sammelstoerung -- ;%{SE}%MKUKATPVW %CVW_COM %VCOMMENT %P 2:-- RSK Sammelstoerung --, 3: VW_COMMENT
      ;ENDFOLD
      ;FOLD F329 = T7 + T9 + F325 ;%{SE}%MKUKATPVW %CVW_SPS %VBOASG %P 2:F329 = T7 + T9 + F325, 3: BOASG
         $FLAG[329] = $TIMER_FLAG[7] OR $TIMER_FLAG[9] OR $FLAG[325]
      ;ENDFOLD
      ;FOLD -- Hilfsflag Startfraesen -- ;%{SE}%MKUKATPVW %CVW_COM %VCOMMENT %P 2:-- Hilfsflag Startfraesen --, 3: VW_COMMENT
      ;ENDFOLD
      ;FOLD F96 = F96 & F287 ;%{SE}%MKUKATPVW %CVW_SPS %VBOASG %P 2:F96 = F96 & F287, 3: BOASG
         $FLAG[96] = $FLAG[96] AND $FLAG[287]
      ;ENDFOLD
      ;FOLD F96 = (F96 & F78 + F98 & F79) & F287 ;%{SE}%MKUKATPVW %CVW_SPS %VBOASG %P 2:F96 = (F96 & F78 + F98 & F79) & F287, 3: BOASG
         $FLAG[96] = ($FLAG[96] AND $FLAG[78] OR $FLAG[98] AND $FLAG[79]) AND $FLAG[287]
      ;ENDFOLD
      ;FOLD F98 = !F130 & F98 + F130 & F287 & F98 ;%{SE}%MKUKATPVW %CVW_SPS %VBOASG %P 2:F98 = !F130 & F98 + F130 & F287 & F98, 3: BOASG
         $FLAG[98] = NOT $FLAG[130] AND $FLAG[98] OR $FLAG[130] AND $FLAG[287] AND $FLAG[98]
      ;ENDFOLD
      ;FOLD F287 = F78 + F79 & F130 ;%{SE}%MKUKATPVW %CVW_SPS %VBOASG %P 2:F287 = F78 + F79 & F130, 3: BOASG
         $FLAG[287] = $FLAG[78] OR $FLAG[79] AND $FLAG[130]
      ;ENDFOLD
      ;FOLD -- Neues Fraesprogramm und Zaehler ruecksetzen -- ;%{SE}%MKUKATPVW %CVW_COM %VCOMMENT %P 2:-- Neues Fraesprogramm und Zaehler ruecksetzen --, 3: VW_COMMENT
      ;ENDFOLD
      ;FOLD bin3 ( F130 ) = 36 ;%{SE}%MKUKATPVW %CVW_SPS %VARIASG %P 2:bin3 ( F130 ) = 36, 3: ARIASG
         VW(#BINOUT,$FLAG[130],3,36)
      ;ENDFOLD
      ;FOLD i4 ( F96 ) = i45 ;%{SE}%MKUKATPVW %CVW_SPS %VARIASG %P 2:i4 ( F96 ) = i45, 3: ARIASG
         VW(#COUNTER,$FLAG[96],4,$COUNT_I[45])
      ;ENDFOLD
      ;FOLD -- Wiederholung beim Startfraesen -- ;%{SE}%MKUKATPVW %CVW_COM %VCOMMENT %P 2:-- Wiederholung beim Startfraesen --, 3: VW_COMMENT
      ;ENDFOLD
      ;FOLD Schritt 58 = E717 & !E718 & (F78 & !F96 + F79 & F130 & !F96) & !F329 & A4039 ;%{SE}%MKUKATPVW %CVW_SPS %VST_CON %P 2:Schritt 58 = E717 & !E718 & (F78 & !F96 + F79 & F130 & !F96) & !F329 & A4039, 3: ST_CON
         IF $IN[717] AND NOT $IN[718] AND ($FLAG[78] AND NOT $FLAG[96] OR $FLAG[79] AND $FLAG[130] AND NOT $FLAG[96]) AND NOT $FLAG[329] AND $OUT[4039] THEN
            PREVSTEP = $APP_INT[5]
            $APP_INT[5] = 58
         ENDIF
      ;ENDFOLD
      ;FOLD -- Weiter wenn Fraesen fertig -- ;%{SE}%MKUKATPVW %CVW_COM %VCOMMENT %P 2:-- Weiter wenn Fraesen fertig --, 3: VW_COMMENT
      ;ENDFOLD
      ;FOLD Schritt 62 = E717 & !E718 & (F79 & F98 & (!F130 + F96) + F78 & F96 + F329 + F325) & A4039 ;%{SE}%MKUKATPVW %CVW_SPS %VST_CON %P 2:Schritt 62 = E717 & !E718 & (F79 & F98 & (!F130 + F96) + F78 & F96 + F329 + F325) & A4039, 3: ST_CON
         IF $IN[717] AND NOT $IN[718] AND ($FLAG[79] AND $FLAG[98] AND (NOT $FLAG[130] OR $FLAG[96]) OR $FLAG[78] AND $FLAG[96] OR $FLAG[329] OR $FLAG[325]) AND $OUT[4039] THEN
            PREVSTEP = $APP_INT[5]
            $APP_INT[5] = 62
         ENDIF
      ;ENDFOLD
   ;ENDFOLD
   ;FOLD SCHRITT 62 -- STAT EZ1/SP1/KE1-- ;%{P}%MKUKATPVW,%CSTEP,%VST_NR,%P 1:SCHRITT, 2:62, 3: STAT EZ1/SP1/KE1
      ;FOLD ;%{H}
         Case 62
      ;ENDFOLD
      ;FOLD F324 = AUS ;%{SE}%MKUKATPVW %CVW_SPS %VBOASG %P 2:F324 = AUS, 3: BOASG
         $FLAG[324] = FALSE
      ;ENDFOLD
      ;FOLD A717 = AUS ;%{SE}%MKUKATPVW %CVW_SPS %VBOASG %P 2:A717 = AUS, 3: BOASG
         $OUT[717] = FALSE
      ;ENDFOLD
      ;FOLD -- KF1 abschalten -- ;%{SE}%MKUKATPVW %CVW_COM %VCOMMENT %P 2:-- KF1 abschalten --, 3: VW_COMMENT
      ;ENDFOLD
      ;FOLD A834 = AUS ;%{SE}%MKUKATPVW %CVW_SPS %VBOASG %P 2:A834 = AUS, 3: BOASG
         $OUT[834] = FALSE
      ;ENDFOLD
      ;FOLD -- Ueberwachungszeit KF1 Versetzeinheit -- ;%{SE}%MKUKATPVW %CVW_COM %VCOMMENT %P 2:-- Ueberwachungszeit KF1 Versetzeinheit --, 3: VW_COMMENT
      ;ENDFOLD
      ;FOLD t8 ( EIN ) = -40[1/10Sek] ;%{SE}%MKUKATPVW %CVW_SPS %VTASG %P 2:t8 ( EIN ) = -40[1/10Sek], 3: TASG
         VW(#SET_TIME,TRUE,8,0,-40)
      ;ENDFOLD
      ;FOLD Schritt 63 = A4039 ;%{SE}%MKUKATPVW %CVW_SPS %VST_CON %P 2:Schritt 63 = A4039, 3: ST_CON
         IF $OUT[4039] THEN
            PREVSTEP = $APP_INT[5]
            $APP_INT[5] = 63
         ENDIF
      ;ENDFOLD
   ;ENDFOLD
   ;FOLD SCHRITT 63 -- STAT EZ1/SP1/KE1 -- ;%{P}%MKUKATPVW,%CSTEP,%VST_NR,%P 1:SCHRITT, 2:63, 3: STAT EZ1/SP1/KE1
      ;FOLD ;%{H}
         Case 63
      ;ENDFOLD
      ;FOLD F328 = AUS ;%{SE}%MKUKATPVW %CVW_SPS %VBOASG %P 2:F328 = AUS, 3: BOASG
         $FLAG[328] = FALSE
      ;ENDFOLD
      ;FOLD -- KF1 Versetzeinheit vor -- ;%{SE}%MKUKATPVW %CVW_COM %VCOMMENT %P 2:-- KF1 Versetzeinheit vor --, 3: VW_COMMENT
      ;ENDFOLD
      ;FOLD A835 = F564 ;%{SE}%MKUKATPVW %CVW_SPS %VBOASG %P 2:A835 = F564, 3: BOASG
         $OUT[835] = $FLAG[564]
      ;ENDFOLD
      ;FOLD -- RSK Fehlerausgabe KS1 Arbeitsst. -- ;%{SE}%MKUKATPVW %CVW_COM %VCOMMENT %P 2:-- RSK Fehlerausgabe KS1 Arbeitsst. --, 3: VW_COMMENT
      ;ENDFOLD
      ;FOLD F324 = (E836 + !E837 + !E838 + E839) & !F323 & !F328 + F324 ;%{SE}%MKUKATPVW %CVW_SPS %VBOASG %P 2:F324 = (E836 + !E837 + !E838 + E839) & !F323 & !F328 + F324, 3: BOASG
         $FLAG[324] = ($IN[836] OR NOT $IN[837] OR NOT $IN[838] OR $IN[839]) AND NOT $FLAG[323] AND NOT $FLAG[328] OR $FLAG[324]
      ;ENDFOLD
      ;FOLD -- RSK Sammelstoerung -- ;%{SE}%MKUKATPVW %CVW_COM %VCOMMENT %P 2:-- RSK Sammelstoerung --, 3: VW_COMMENT
      ;ENDFOLD
      ;FOLD F329 = F324 + F325 ;%{SE}%MKUKATPVW %CVW_SPS %VBOASG %P 2:F329 = F324 + F325, 3: BOASG
         $FLAG[329] = $FLAG[324] OR $FLAG[325]
      ;ENDFOLD
      ;FOLD -- Ueberwachungszeit KS1 schwenken -- ;%{SE}%MKUKATPVW %CVW_COM %VCOMMENT %P 2:-- Ueberwachungszeit KS1 schwenken --, 3: VW_COMMENT
      ;ENDFOLD
      ;FOLD t9 ( EIN ) = -100[1/10Sek] ;%{SE}%MKUKATPVW %CVW_SPS %VTASG %P 2:t9 ( EIN ) = -100[1/10Sek], 3: TASG
         VW(#SET_TIME,TRUE,9,0,-100)
      ;ENDFOLD
      ;FOLD Schritt 62 = F324 & (E26 + E27) & A4039 ;%{SE}%MKUKATPVW %CVW_SPS %VST_CON %P 2:Schritt 62 = F324 & (E26 + E27) & A4039, 3: ST_CON
         IF $FLAG[324] AND ($IN[26] OR $IN[27]) AND $OUT[4039] THEN
            PREVSTEP = $APP_INT[5]
            $APP_INT[5] = 62
         ENDIF
      ;ENDFOLD
      ;FOLD Schritt 64 = (!F324 & (E835 & F564 + !E835 & !F564) + T8 + F325) & A4039 ;%{SE}%MKUKATPVW %CVW_SPS %VST_CON %P 2:Schritt 64 = (!F324 & (E835 & F564 + !E835 & !F564) + T8 + F325) & A4039, 3: ST_CON
         IF (NOT $FLAG[324] AND ($IN[835] AND $FLAG[564] OR NOT $IN[835] AND NOT $FLAG[564]) OR $TIMER_FLAG[8] OR $FLAG[325]) AND $OUT[4039] THEN
            PREVSTEP = $APP_INT[5]
            $APP_INT[5] = 64
         ENDIF
      ;ENDFOLD
   ;ENDFOLD
   ;FOLD SCHRITT 64 -- STAT EZ1/SP1/KE1-- ;%{P}%MKUKATPVW,%CSTEP,%VST_NR,%P 1:SCHRITT, 2:64, 3: STAT EZ1/SP1/KE1
      ;FOLD ;%{H}
         Case 64
      ;ENDFOLD
      ;FOLD F323 = AUS ;%{SE}%MKUKATPVW %CVW_SPS %VBOASG %P 2:F323 = AUS, 3: BOASG
         $FLAG[323] = FALSE
      ;ENDFOLD
      ;FOLD F328 = AUS ;%{SE}%MKUKATPVW %CVW_SPS %VBOASG %P 2:F328 = AUS, 3: BOASG
         $FLAG[328] = FALSE
      ;ENDFOLD
      ;FOLD -- RSK Sammelstoerung -- ;%{SE}%MKUKATPVW %CVW_COM %VCOMMENT %P 2:-- RSK Sammelstoerung --, 3: VW_COMMENT
      ;ENDFOLD
      ;FOLD F329 = F325 ;%{SE}%MKUKATPVW %CVW_SPS %VBOASG %P 2:F329 = F325, 3: BOASG
         $FLAG[329] = $FLAG[325]
      ;ENDFOLD
      ;FOLD -- KF1 ein -- ;%{SE}%MKUKATPVW %CVW_COM %VCOMMENT %P 2:-- KF1 ein --, 3: VW_COMMENT
      ;ENDFOLD
      ;FOLD A834 = EIN ;%{SE}%MKUKATPVW %CVW_SPS %VBOASG %P 2:A834 = EIN, 3: BOASG
         $OUT[834] = TRUE
      ;ENDFOLD
      ;FOLD -- KS1 in Ruhestellung schwenken -- ;%{SE}%MKUKATPVW %CVW_COM %VCOMMENT %P 2:-- KS1 in Ruhestellung schwenken --, 3: VW_COMMENT
      ;ENDFOLD
      ;FOLD A840 = (F745 + !F714) & E717 & (E835 & F564 + !E835 & !F564) ;%{SE}%MKUKATPVW %CVW_SPS %VBOASG %P 2:A840 = (F745 + !F714) & E717 & (E835 & F564 + !E835 & !F564), 3: BOASG
         $OUT[840] = ($FLAG[745] OR NOT $FLAG[714]) AND $IN[717] AND ($IN[835] AND $FLAG[564] OR NOT $IN[835] AND NOT $FLAG[564])
      ;ENDFOLD
      ;FOLD Schritt 65 = (F745 + !F714 + T9) & (A840 + T9) & E717 & A4039 ;%{SE}%MKUKATPVW %CVW_SPS %VST_CON %P 2:Schritt 65 = (F745 + !F714 + T9) & (A840 + T9) & E717 & A4039, 3: ST_CON
         IF ($FLAG[745] OR NOT $FLAG[714] OR $TIMER_FLAG[9]) AND ($OUT[840] OR $TIMER_FLAG[9]) AND $IN[717] AND $OUT[4039] THEN
            PREVSTEP = $APP_INT[5]
            $APP_INT[5] = 65
         ENDIF
      ;ENDFOLD
   ;ENDFOLD
   ;FOLD SCHRITT 65 -- STAT EZ1/SP1/KE1 -- ;%{P}%MKUKATPVW,%CSTEP,%VST_NR,%P 1:SCHRITT, 2:65, 3: STAT EZ1/SP1/KE1
      ;FOLD ;%{H}
         Case 65
      ;ENDFOLD
      ;FOLD -- Hilfsflag SK Programmwechsel -- ;%{SE}%MKUKATPVW %CVW_COM %VCOMMENT %P 2:-- Hilfsflag SK Programmwechsel --, 3: VW_COMMENT
      ;ENDFOLD
      ;FOLD F334 = AUS ;%{SE}%MKUKATPVW %CVW_SPS %VBOASG %P 2:F334 = AUS, 3: BOASG
         $FLAG[334] = FALSE
      ;ENDFOLD
      ;FOLD -- RSK Fehlerausgabe KF Versetzeinheit -- ;%{SE}%MKUKATPVW %CVW_COM %VCOMMENT %P 2:-- RSK Fehlerausgabe KF Versetzeinheit --, 3: VW_COMMENT
      ;ENDFOLD
      ;FOLD F328 = !E835 & F564 & !F323 + F328 ;%{SE}%MKUKATPVW %CVW_SPS %VBOASG %P 2:F328 = !E835 & F564 & !F323 + F328, 3: BOASG
         $FLAG[328] = NOT $IN[835] AND $FLAG[564] AND NOT $FLAG[323] OR $FLAG[328]
      ;ENDFOLD
      ;FOLD -- RSK Fehlerausgabe KS1 Ruhestellung -- ;%{SE}%MKUKATPVW %CVW_COM %VCOMMENT %P 2:-- RSK Fehlerausgabe KS1 Ruhestellung --, 3: VW_COMMENT
      ;ENDFOLD
      ;FOLD F323 = (!E836 + E837 + E838 + !E839) & T9 & (E835 + !F564) + F323 ;%{SE}%MKUKATPVW %CVW_SPS %VBOASG %P 2:F323 = (!E836 + E837 + E838 + !E839) & T9 & (E835 + !F564) + F323, 3: BOASG
         $FLAG[323] = (NOT $IN[836] OR $IN[837] OR $IN[838] OR NOT $IN[839]) AND $TIMER_FLAG[9] AND ($IN[835] OR NOT $FLAG[564]) OR $FLAG[323]
      ;ENDFOLD
      ;FOLD -- RSK Fehlerausgabe EZ/SP min. Oeffnung -- ;%{SE}%MKUKATPVW %CVW_COM %VCOMMENT %P 2:-- RSK Fehlerausgabe EZ/SP min. Oeffnung --, 3: VW_COMMENT
      ;ENDFOLD
      ;FOLD F333 = !F745 ;%{SE}%MKUKATPVW %CVW_SPS %VBOASG %P 2:F333 = !F745, 3: BOASG
         $FLAG[333] = NOT $FLAG[745]
      ;ENDFOLD
      ;FOLD -- RSK Sammelstoerung -- ;%{SE}%MKUKATPVW %CVW_COM %VCOMMENT %P 2:-- RSK Sammelstoerung --, 3: VW_COMMENT
      ;ENDFOLD
      ;FOLD F329 = F323 + F325 + F328 + F333 ;%{SE}%MKUKATPVW %CVW_SPS %VBOASG %P 2:F329 = F323 + F325 + F328 + F333, 3: BOASG
         $FLAG[329] = $FLAG[323] OR $FLAG[325] OR $FLAG[328] OR $FLAG[333]
      ;ENDFOLD
      ;FOLD A834 = !F323 & !F328 ;%{SE}%MKUKATPVW %CVW_SPS %VBOASG %P 2:A834 = !F323 & !F328, 3: BOASG
         $OUT[834] = NOT $FLAG[323] AND NOT $FLAG[328]
      ;ENDFOLD
      ;FOLD A836 = F564 ;%{SE}%MKUKATPVW %CVW_SPS %VBOASG %P 2:A836 = F564, 3: BOASG
         $OUT[836] = $FLAG[564]
      ;ENDFOLD
      ;FOLD Schritt 63 = (F323 + F328) & (E26 + E27) & A4039 ;%{SE}%MKUKATPVW %CVW_SPS %VST_CON %P 2:Schritt 63 = (F323 + F328) & (E26 + E27) & A4039, 3: ST_CON
         IF ($FLAG[323] OR $FLAG[328]) AND ($IN[26] OR $IN[27]) AND $OUT[4039] THEN
            PREVSTEP = $APP_INT[5]
            $APP_INT[5] = 63
         ENDIF
      ;ENDFOLD
      ;FOLD Schritt 66 = !A840 & E836 & !E837 & !E838 & E839 & A4039 ;%{SE}%MKUKATPVW %CVW_SPS %VST_CON %P 2:Schritt 66 = !A840 & E836 & !E837 & !E838 & E839 & A4039, 3: ST_CON
         IF NOT $OUT[840] AND $IN[836] AND NOT $IN[837] AND NOT $IN[838] AND $IN[839] AND $OUT[4039] THEN
            PREVSTEP = $APP_INT[5]
            $APP_INT[5] = 66
         ENDIF
      ;ENDFOLD
   ;ENDFOLD
   ;FOLD SCHRITT 66 -- STAT EZ1/SP1/KE1 -- ;%{P}%MKUKATPVW,%CSTEP,%VST_NR,%P 1:SCHRITT, 2:66, 3: STAT EZ1/SP1/KE1
      ;FOLD ;%{H}
         Case 66
      ;ENDFOLD
      ;FOLD F323 = AUS ;%{SE}%MKUKATPVW %CVW_SPS %VBOASG %P 2:F323 = AUS, 3: BOASG
         $FLAG[323] = FALSE
      ;ENDFOLD
      ;FOLD F328 = AUS ;%{SE}%MKUKATPVW %CVW_SPS %VBOASG %P 2:F328 = AUS, 3: BOASG
         $FLAG[328] = FALSE
      ;ENDFOLD
      ;FOLD -- RSK Sammelstoerung -- ;%{SE}%MKUKATPVW %CVW_COM %VCOMMENT %P 2:-- RSK Sammelstoerung --, 3: VW_COMMENT
      ;ENDFOLD
      ;FOLD F329 = F325 ;%{SE}%MKUKATPVW %CVW_SPS %VBOASG %P 2:F329 = F325, 3: BOASG
         $FLAG[329] = $FLAG[325]
      ;ENDFOLD
      ;FOLD t9 ( EIN ) = STOP ;%{SE}%MKUKATPVW %CVW_SPS %VTSTOP %P 2:t9 ( EIN ) = STOP, 3: TSTOP
         VW(#SET_TIME,TRUE,9,1,0)
      ;ENDFOLD
      ;FOLD -- KF1 Versetzeinheit rueck -- ;%{SE}%MKUKATPVW %CVW_COM %VCOMMENT %P 2:-- KF1 Versetzeinheit rueck --, 3: VW_COMMENT
      ;ENDFOLD
      ;FOLD A835 = AUS ;%{SE}%MKUKATPVW %CVW_SPS %VBOASG %P 2:A835 = AUS, 3: BOASG
         $OUT[835] = FALSE
      ;ENDFOLD
      ;FOLD -- KF1 aus -- ;%{SE}%MKUKATPVW %CVW_COM %VCOMMENT %P 2:-- KF1 aus --, 3: VW_COMMENT
      ;ENDFOLD
      ;FOLD A834 = AUS ;%{SE}%MKUKATPVW %CVW_SPS %VBOASG %P 2:A834 = AUS, 3: BOASG
         $OUT[834] = FALSE
      ;ENDFOLD
      ;FOLD -- KF1 Ausblasen -- ;%{SE}%MKUKATPVW %CVW_COM %VCOMMENT %P 2:-- KF1 Ausblasen --, 3: VW_COMMENT
      ;ENDFOLD
      ;FOLD A836 = (F330 + F331 + F332) & F737 ;%{SE}%MKUKATPVW %CVW_SPS %VBOASG %P 2:A836 = (F330 + F331 + F332) & F737, 3: BOASG
         $OUT[836] = ($FLAG[330] OR $FLAG[331] OR $FLAG[332]) AND $FLAG[737]
      ;ENDFOLD
      ;FOLD F168 = !F329 & !F830 ;%{SE}%MKUKATPVW %CVW_SPS %VBOASG %P 2:F168 = !F329 & !F830, 3: BOASG
         $FLAG[168] = NOT $FLAG[329] AND NOT $FLAG[830]
      ;ENDFOLD
      ;FOLD bin1 ( F168 ) = 1 ;%{SE}%MKUKATPVW %CVW_SPS %VARIASG %P 2:bin1 ( F168 ) = 1, 3: ARIASG
         VW(#BINOUT,$FLAG[168],1,1)
      ;ENDFOLD
      ;FOLD F168 = AUS ;%{SE}%MKUKATPVW %CVW_SPS %VBOASG %P 2:F168 = AUS, 3: BOASG
         $FLAG[168] = FALSE
      ;ENDFOLD
      ;FOLD bin3 ( !F329 ) = 1 ;%{SE}%MKUKATPVW %CVW_SPS %VARIASG %P 2:bin3 ( !F329 ) = 1, 3: ARIASG
         VW(#BINOUT,NOT $FLAG[329],3,1)
      ;ENDFOLD
      ;FOLD -- Wartezeit Programmwechsel SK -- ;%{SE}%MKUKATPVW %CVW_COM %VCOMMENT %P 2:-- Wartezeit Programmwechsel SK --, 3: VW_COMMENT
      ;ENDFOLD
      ;FOLD T8 ( !F334 ) = -2[1/10Sek] ;%{SE}%MKUKATPVW %CVW_SPS %VTASG %P 2:T8 ( !F334 ) = -2[1/10Sek], 3: TASG
         VW(#SET_TIME,NOT $FLAG[334],8,0,-2)
      ;ENDFOLD
      ;FOLD -- Hilfsflag SK Programmwechsel -- ;%{SE}%MKUKATPVW %CVW_COM %VCOMMENT %P 2:-- Hilfsflag SK Programmwechsel --, 3: VW_COMMENT
      ;ENDFOLD
      ;FOLD F334 = EIN ;%{SE}%MKUKATPVW %CVW_SPS %VBOASG %P 2:F334 = EIN, 3: BOASG
         $FLAG[334] = TRUE
      ;ENDFOLD
      ;FOLD -- Ueberwachungszeit EZ1/SP1/KE1 SZ1 Messen -- ;%{SE}%MKUKATPVW %CVW_COM %VCOMMENT %P 2:-- Ueberwachungszeit EZ1/SP1/KE1 SZ1 Messen --, 3: VW_COMMENT
      ;ENDFOLD
      ;FOLD t9 ( EIN ) = -150[1/10Sek] ;%{SE}%MKUKATPVW %CVW_SPS %VTASG %P 2:t9 ( EIN ) = -150[1/10Sek], 3: TASG
         VW(#SET_TIME,TRUE,9,0,-150)
      ;ENDFOLD
      ;FOLD Schritt 51 = (F325 + F329) & (E26 + E27) & A4039 ;%{SE}%MKUKATPVW %CVW_SPS %VST_CON %P 2:Schritt 51 = (F325 + F329) & (E26 + E27) & A4039, 3: ST_CON
         IF ($FLAG[325] OR $FLAG[329]) AND ($IN[26] OR $IN[27]) AND $OUT[4039] THEN
            PREVSTEP = $APP_INT[5]
            $APP_INT[5] = 51
         ENDIF
      ;ENDFOLD
      ;FOLD Schritt 67 = T8 & !F325 & !F329 & A4039 ;%{SE}%MKUKATPVW %CVW_SPS %VST_CON %P 2:Schritt 67 = T8 & !F325 & !F329 & A4039, 3: ST_CON
         IF $TIMER_FLAG[8] AND NOT $FLAG[325] AND NOT $FLAG[329] AND $OUT[4039] THEN
            PREVSTEP = $APP_INT[5]
            $APP_INT[5] = 67
         ENDIF
      ;ENDFOLD
   ;ENDFOLD
   ;FOLD SCHRITT 67 -- STAT EZ1/SP1/KE1 -- ;%{P}%MKUKATPVW,%CSTEP,%VST_NR,%P 1:SCHRITT, 2:67, 3: STAT EZ1/SP1/KE1
      ;FOLD ;%{H}
         Case 67
      ;ENDFOLD
      ;FOLD -- Hilfsflag SK Programmwechsel -- ;%{SE}%MKUKATPVW %CVW_COM %VCOMMENT %P 2:-- Hilfsflag SK Programmwechsel --, 3: VW_COMMENT
      ;ENDFOLD
      ;FOLD F334 = AUS ;%{SE}%MKUKATPVW %CVW_SPS %VBOASG %P 2:F334 = AUS, 3: BOASG
         $FLAG[334] = FALSE
      ;ENDFOLD
      ;FOLD -- Quitt. Fraesen SK1 -- ;%{SE}%MKUKATPVW %CVW_COM %VCOMMENT %P 2:-- Quitt. Fraesen SK1 --, 3: VW_COMMENT
      ;ENDFOLD
      ;FOLD A786 = !F329 & !F322 ;%{SE}%MKUKATPVW %CVW_SPS %VBOASG %P 2:A786 = !F329 & !F322, 3: BOASG
         $OUT[786] = NOT $FLAG[329] AND NOT $FLAG[322]
      ;ENDFOLD
      ;FOLD -- RSK Sammelstoerung -- ;%{SE}%MKUKATPVW %CVW_COM %VCOMMENT %P 2:-- RSK Sammelstoerung --, 3: VW_COMMENT
      ;ENDFOLD
      ;FOLD F329 = T9 ;%{SE}%MKUKATPVW %CVW_SPS %VBOASG %P 2:F329 = T9, 3: BOASG
         $FLAG[329] = $TIMER_FLAG[9]
      ;ENDFOLD
      ;FOLD -- Messen nach Fraesen -- ;%{SE}%MKUKATPVW %CVW_COM %VCOMMENT %P 2:-- Messen nach Fraesen --, 3: VW_COMMENT
      ;ENDFOLD
      ;FOLD A759 = !F78 & F79 ;%{SE}%MKUKATPVW %CVW_SPS %VBOASG %P 2:A759 = !F78 & F79, 3: BOASG
         $OUT[759] = NOT $FLAG[78] AND $FLAG[79]
      ;ENDFOLD
      ;FOLD A758 = F78 & !F79 ;%{SE}%MKUKATPVW %CVW_SPS %VBOASG %P 2:A758 = F78 & !F79, 3: BOASG
         $OUT[758] = $FLAG[78] AND NOT $FLAG[79]
      ;ENDFOLD
      ;FOLD A757 = (F78 + F79) & !F329 ;%{SE}%MKUKATPVW %CVW_SPS %VBOASG %P 2:A757 = (F78 + F79) & !F329, 3: BOASG
         $OUT[757] = ($FLAG[78] OR $FLAG[79]) AND NOT $FLAG[329]
      ;ENDFOLD
      ;FOLD Schritt 68 = !E786 & E787 & !E788 & A4039 ;%{SE}%MKUKATPVW %CVW_SPS %VST_CON %P 2:Schritt 68 = !E786 & E787 & !E788 & A4039, 3: ST_CON
         IF NOT $IN[786] AND $IN[787] AND NOT $IN[788] AND $OUT[4039] THEN
            PREVSTEP = $APP_INT[5]
            $APP_INT[5] = 68
         ENDIF
      ;ENDFOLD
   ;ENDFOLD
   ;FOLD SCHRITT 68 -- STAT EZ1/SP1/KE1 -- ;%{P}%MKUKATPVW,%CSTEP,%VST_NR,%P 1:SCHRITT, 2:68, 3: STAT EZ1/SP1/KE1
      ;FOLD ;%{H}
         Case 68
      ;ENDFOLD
      ;FOLD -- Hilfsflag SK Programmwechsel -- ;%{SE}%MKUKATPVW %CVW_COM %VCOMMENT %P 2:-- Hilfsflag SK Programmwechsel --, 3: VW_COMMENT
      ;ENDFOLD
      ;FOLD F334 = AUS ;%{SE}%MKUKATPVW %CVW_SPS %VBOASG %P 2:F334 = AUS, 3: BOASG
         $FLAG[334] = FALSE
      ;ENDFOLD
      ;FOLD -- RSK Sammelstoerung -- ;%{SE}%MKUKATPVW %CVW_COM %VCOMMENT %P 2:-- RSK Sammelstoerung --, 3: VW_COMMENT
      ;ENDFOLD
      ;FOLD F329 = T9 ;%{SE}%MKUKATPVW %CVW_SPS %VBOASG %P 2:F329 = T9, 3: BOASG
         $FLAG[329] = $TIMER_FLAG[9]
      ;ENDFOLD
      ;FOLD Schritt 69 = E717 & (E757 & !E776 + T9) & A4039 ;%{SE}%MKUKATPVW %CVW_SPS %VST_CON %P 2:Schritt 69 = E717 & (E757 & !E776 + T9) & A4039, 3: ST_CON
         IF $IN[717] AND ($IN[757] AND NOT $IN[776] OR $TIMER_FLAG[9]) AND $OUT[4039] THEN
            PREVSTEP = $APP_INT[5]
            $APP_INT[5] = 69
         ENDIF
      ;ENDFOLD
   ;ENDFOLD
   ;FOLD SCHRITT 69 -- STAT EZ1/SP1/KE1-- ;%{P}%MKUKATPVW,%CSTEP,%VST_NR,%P 1:SCHRITT, 2:69, 3: STAT EZ1/SP1/KE1
      ;FOLD ;%{H}
         Case 69
      ;ENDFOLD
      ;FOLD -- RSK Fehlerausgabe Kappenverschleiss -- ;%{SE}%MKUKATPVW %CVW_COM %VCOMMENT %P 2:-- RSK Fehlerausgabe Kappenverschleiss --, 3: VW_COMMENT
      ;ENDFOLD
      ;FOLD F122 = E777 ;%{SE}%MKUKATPVW %CVW_SPS %VBOASG %P 2:F122 = E777, 3: BOASG
         $FLAG[122] = $IN[777]
      ;ENDFOLD
      ;FOLD -- RSK Fehlerausgabe Messen -- ;%{SE}%MKUKATPVW %CVW_COM %VCOMMENT %P 2:-- RSK Fehlerausgabe Messen --, 3: VW_COMMENT
      ;ENDFOLD
      ;FOLD F326 = E776 + E777 + E778 + F326 ;%{SE}%MKUKATPVW %CVW_SPS %VBOASG %P 2:F326 = E776 + E777 + E778 + F326, 3: BOASG
         $FLAG[326] = $IN[776] OR $IN[777] OR $IN[778] OR $FLAG[326]
      ;ENDFOLD
      ;FOLD -- RSK Sammelstoerung -- ;%{SE}%MKUKATPVW %CVW_COM %VCOMMENT %P 2:-- RSK Sammelstoerung --, 3: VW_COMMENT
      ;ENDFOLD
      ;FOLD F329 = F326 ;%{SE}%MKUKATPVW %CVW_SPS %VBOASG %P 2:F329 = F326, 3: BOASG
         $FLAG[329] = $FLAG[326]
      ;ENDFOLD
      ;FOLD A758 = AUS ;%{SE}%MKUKATPVW %CVW_SPS %VBOASG %P 2:A758 = AUS, 3: BOASG
         $OUT[758] = FALSE
      ;ENDFOLD
      ;FOLD A759 = AUS ;%{SE}%MKUKATPVW %CVW_SPS %VBOASG %P 2:A759 = AUS, 3: BOASG
         $OUT[759] = FALSE
      ;ENDFOLD
      ;FOLD -- Ueberwachungszeit EZ1/SP1/KE1 Setzhub 2 -- ;%{SE}%MKUKATPVW %CVW_COM %VCOMMENT %P 2:-- Ueberwachungszeit EZ1/SP1/KE1 Setzhub 2 --, 3: VW_COMMENT
      ;ENDFOLD
      ;FOLD t9 ( EIN ) = -80[1/10Sek] ;%{SE}%MKUKATPVW %CVW_SPS %VTASG %P 2:t9 ( EIN ) = -80[1/10Sek], 3: TASG
         VW(#SET_TIME,TRUE,9,0,-80)
      ;ENDFOLD
      ;FOLD -- Druckvorgabe SK1/EZ1/SP1/KE1 -- ;%{SE}%MKUKATPVW %CVW_COM %VCOMMENT %P 2:-- Druckvorgabe SK1/EZ1/SP1/KE1 --, 3: VW_COMMENT
      ;ENDFOLD
      ;FOLD F168 = F78 & !F830 ;%{SE}%MKUKATPVW %CVW_SPS %VBOASG %P 2:F168 = F78 & !F830, 3: BOASG
         $FLAG[168] = $FLAG[78] AND NOT $FLAG[830]
      ;ENDFOLD
      ;FOLD bin1 ( F168 ) = 41 ;%{SE}%MKUKATPVW %CVW_SPS %VARIASG %P 2:bin1 ( F168 ) = 41, 3: ARIASG
         VW(#BINOUT,$FLAG[168],1,41)
      ;ENDFOLD
      ;FOLD F168 = F79 & !F830 ;%{SE}%MKUKATPVW %CVW_SPS %VBOASG %P 2:F168 = F79 & !F830, 3: BOASG
         $FLAG[168] = $FLAG[79] AND NOT $FLAG[830]
      ;ENDFOLD
      ;FOLD bin1 ( F168 ) = 51 ;%{SE}%MKUKATPVW %CVW_SPS %VARIASG %P 2:bin1 ( F168 ) = 51, 3: ARIASG
         VW(#BINOUT,$FLAG[168],1,51)
      ;ENDFOLD
      ;FOLD F168 = AUS ;%{SE}%MKUKATPVW %CVW_SPS %VBOASG %P 2:F168 = AUS, 3: BOASG
         $FLAG[168] = FALSE
      ;ENDFOLD
      ;FOLD bin3 ( F78 ) = 41 ;%{SE}%MKUKATPVW %CVW_SPS %VARIASG %P 2:bin3 ( F78 ) = 41, 3: ARIASG
         VW(#BINOUT,$FLAG[78],3,41)
      ;ENDFOLD
      ;FOLD bin3 ( F79 ) = 51 ;%{SE}%MKUKATPVW %CVW_SPS %VARIASG %P 2:bin3 ( F79 ) = 51, 3: ARIASG
         VW(#BINOUT,$FLAG[79],3,51)
      ;ENDFOLD
      ;FOLD -- Wartezeit Programmwechsel SK -- ;%{SE}%MKUKATPVW %CVW_COM %VCOMMENT %P 2:-- Wartezeit Programmwechsel SK --, 3: VW_COMMENT
      ;ENDFOLD
      ;FOLD T8 ( !F334 ) = -2[1/10Sek] ;%{SE}%MKUKATPVW %CVW_SPS %VTASG %P 2:T8 ( !F334 ) = -2[1/10Sek], 3: TASG
         VW(#SET_TIME,NOT $FLAG[334],8,0,-2)
      ;ENDFOLD
      ;FOLD -- Hilfsflag SK Programmwechsel -- ;%{SE}%MKUKATPVW %CVW_COM %VCOMMENT %P 2:-- Hilfsflag SK Programmwechsel --, 3: VW_COMMENT
      ;ENDFOLD
      ;FOLD F334 = EIN ;%{SE}%MKUKATPVW %CVW_SPS %VBOASG %P 2:F334 = EIN, 3: BOASG
         $FLAG[334] = TRUE
      ;ENDFOLD
      ;FOLD Schritt 70 = T8 & !F335 & A4039 ;%{SE}%MKUKATPVW %CVW_SPS %VST_CON %P 2:Schritt 70 = T8 & !F335 & A4039, 3: ST_CON
         IF $TIMER_FLAG[8] AND NOT $FLAG[335] AND $OUT[4039] THEN
            PREVSTEP = $APP_INT[5]
            $APP_INT[5] = 70
         ENDIF
      ;ENDFOLD
      ;FOLD Schritt 70 = T8 & F335 & !F78 & A4039 ;%{SE}%MKUKATPVW %CVW_SPS %VST_CON %P 2:Schritt 70 = T8 & F335 & !F78 & A4039, 3: ST_CON
         IF $TIMER_FLAG[8] AND $FLAG[335] AND NOT $FLAG[78] AND $OUT[4039] THEN
            PREVSTEP = $APP_INT[5]
            $APP_INT[5] = 70
         ENDIF
      ;ENDFOLD
      ;FOLD Schritt 217 = T8 & F335 & F78 & A4039 ;%{SE}%MKUKATPVW %CVW_SPS %VST_CON %P 2:Schritt 217 = T8 & F335 & F78 & A4039, 3: ST_CON
         IF $TIMER_FLAG[8] AND $FLAG[335] AND $FLAG[78] AND $OUT[4039] THEN
            PREVSTEP = $APP_INT[5]
            $APP_INT[5] = 217
         ENDIF
      ;ENDFOLD
   ;ENDFOLD
   ;FOLD SCHRITT 70 -- STAT EZ1/SP1/KE1 -- ;%{P}%MKUKATPVW,%CSTEP,%VST_NR,%P 1:SCHRITT, 2:70, 3: STAT EZ1/SP1/KE1
      ;FOLD ;%{H}
         Case 70
      ;ENDFOLD
      ;FOLD -- Hilfsflag SK Programmwechsel -- ;%{SE}%MKUKATPVW %CVW_COM %VCOMMENT %P 2:-- Hilfsflag SK Programmwechsel --, 3: VW_COMMENT
      ;ENDFOLD
      ;FOLD F334 = AUS ;%{SE}%MKUKATPVW %CVW_SPS %VBOASG %P 2:F334 = AUS, 3: BOASG
         $FLAG[334] = FALSE
      ;ENDFOLD
      ;FOLD A757 = AUS ;%{SE}%MKUKATPVW %CVW_SPS %VBOASG %P 2:A757 = AUS, 3: BOASG
         $OUT[757] = FALSE
      ;ENDFOLD
      ;FOLD -- EZ1/SP1/KE1 schliessen -- ;%{SE}%MKUKATPVW %CVW_COM %VCOMMENT %P 2:-- EZ1/SP1/KE1 schliessen --, 3: VW_COMMENT
      ;ENDFOLD
      ;FOLD A717 = AUS ;%{SE}%MKUKATPVW %CVW_SPS %VBOASG %P 2:A717 = AUS, 3: BOASG
         $OUT[717] = FALSE
      ;ENDFOLD
      ;FOLD A718 = !F329 & !F122 ;%{SE}%MKUKATPVW %CVW_SPS %VBOASG %P 2:A718 = !F329 & !F122, 3: BOASG
         $OUT[718] = NOT $FLAG[329] AND NOT $FLAG[122]
      ;ENDFOLD
      ;FOLD -- Ueberwachungszeit Kurzschlussschweissung SK1 -- ;%{SE}%MKUKATPVW %CVW_COM %VCOMMENT %P 2:-- Ueberwachungszeit Kurzschlussschweissung SK1 --, 3: VW_COMMENT
      ;ENDFOLD
      ;FOLD t9 ( EIN ) = -80[1/10Sek] ;%{SE}%MKUKATPVW %CVW_SPS %VTASG %P 2:t9 ( EIN ) = -80[1/10Sek], 3: TASG
         VW(#SET_TIME,TRUE,9,0,-80)
      ;ENDFOLD
      ;FOLD Schritt 71 = T8 & !E717 & E718 + E717 & !E718 & (F329 + F326 + F122) & A4039 ;%{SE}%MKUKATPVW %CVW_SPS %VST_CON %P 2:Schritt 71 = T8 & !E717 & E718 + E717 & !E718 & (F329 + F326 + F122) & A4039, 3: ST_CON
         IF $TIMER_FLAG[8] AND NOT $IN[717] AND $IN[718] OR $IN[717] AND NOT $IN[718] AND ($FLAG[329] OR $FLAG[326] OR $FLAG[122]) AND $OUT[4039] THEN
            PREVSTEP = $APP_INT[5]
            $APP_INT[5] = 71
         ENDIF
      ;ENDFOLD
   ;ENDFOLD
   ;FOLD SCHRITT 71 -- STAT EZ1/SP1/KE1-- ;%{P}%MKUKATPVW,%CSTEP,%VST_NR,%P 1:SCHRITT, 2:71, 3: STAT EZ1/SP1/KE1
      ;FOLD ;%{H}
         Case 71
      ;ENDFOLD
      ;FOLD -- Hilfsflag SK Programmwechsel -- ;%{SE}%MKUKATPVW %CVW_COM %VCOMMENT %P 2:-- Hilfsflag SK Programmwechsel --, 3: VW_COMMENT
      ;ENDFOLD
      ;FOLD F334 = AUS ;%{SE}%MKUKATPVW %CVW_SPS %VBOASG %P 2:F334 = AUS, 3: BOASG
         $FLAG[334] = FALSE
      ;ENDFOLD
      ;FOLD t9 ( EIN ) = STOP ;%{SE}%MKUKATPVW %CVW_SPS %VTSTOP %P 2:t9 ( EIN ) = STOP, 3: TSTOP
         VW(#SET_TIME,TRUE,9,1,0)
      ;ENDFOLD
      ;FOLD -- RSK Fehlerausgabe Kraftaufbau -- ;%{SE}%MKUKATPVW %CVW_COM %VCOMMENT %P 2:-- RSK Fehlerausgabe Kraftaufbau --, 3: VW_COMMENT
      ;ENDFOLD
      ;FOLD F325 = T9 + F325 ;%{SE}%MKUKATPVW %CVW_SPS %VBOASG %P 2:F325 = T9 + F325, 3: BOASG
         $FLAG[325] = $TIMER_FLAG[9] OR $FLAG[325]
      ;ENDFOLD
      ;FOLD -- RSK Fehlerausgabe K -- ;%{SE}%MKUKATPVW %CVW_COM %VCOMMENT %P 2:-- RSK Fehlerausgabe K --, 3: VW_COMMENT
      ;ENDFOLD
      ;FOLD F327 = (A785 & !F830 + A718 & F830) & (E805 + !E802) + F327 ;%{SE}%MKUKATPVW %CVW_SPS %VBOASG %P 2:F327 = (A785 & !F830 + A718 & F830) & (E805 + !E802) + F327, 3: BOASG
         $FLAG[327] = ($OUT[785] AND NOT $FLAG[830] OR $OUT[718] AND $FLAG[830]) AND ($IN[805] OR NOT $IN[802]) OR $FLAG[327]
      ;ENDFOLD
      ;FOLD -- RSK Sammelstoerung -- ;%{SE}%MKUKATPVW %CVW_COM %VCOMMENT %P 2:-- RSK Sammelstoerung --, 3: VW_COMMENT
      ;ENDFOLD
      ;FOLD F329 = F325 + F326 + F327 ;%{SE}%MKUKATPVW %CVW_SPS %VBOASG %P 2:F329 = F325 + F326 + F327, 3: BOASG
         $FLAG[329] = $FLAG[325] OR $FLAG[326] OR $FLAG[327]
      ;ENDFOLD
      ;FOLD -- Kurzschlussschweissung SK1 -- ;%{SE}%MKUKATPVW %CVW_COM %VCOMMENT %P 2:-- Kurzschlussschweissung SK1 --, 3: VW_COMMENT
      ;ENDFOLD
      ;FOLD A785 = !F325 & !F329 & !F122 & !F830 ;%{SE}%MKUKATPVW %CVW_SPS %VBOASG %P 2:A785 = !F325 & !F329 & !F122 & !F830, 3: BOASG
         $OUT[785] = NOT $FLAG[325] AND NOT $FLAG[329] AND NOT $FLAG[122] AND NOT $FLAG[830]
      ;ENDFOLD
      ;FOLD -- Flagbildung Wiederholfraesen -- ;%{SE}%MKUKATPVW %CVW_COM %VCOMMENT %P 2:-- Flagbildung Wiederholfraesen --, 3: VW_COMMENT
      ;ENDFOLD
      ;FOLD F749 = (F322 + F323 + F325 + F326 + F327 + F329) & !F748 ;%{SE}%MKUKATPVW %CVW_SPS %VBOASG %P 2:F749 = (F322 + F323 + F325 + F326 + F327 + F329) & !F748, 3: BOASG
         $FLAG[749] = ($FLAG[322] OR $FLAG[323] OR $FLAG[325] OR $FLAG[326] OR $FLAG[327] OR $FLAG[329]) AND NOT $FLAG[748]
      ;ENDFOLD
      ;FOLD Schritt 51 = E717 & !E718 & (F322 + F323 + F325 + F326 + F327 + F329) & (E26 + E27) & A4039 ;%{SE}%MKUKATPVW %CVW_SPS %VST_CON %P 2:Schritt 51 = E717 & !E718 & (F322 + F323 + F325 + F326 + F327 + F329) & (E26 + E27) & A4039, 3: ST_CON
         IF $IN[717] AND NOT $IN[718] AND ($FLAG[322] OR $FLAG[323] OR $FLAG[325] OR $FLAG[326] OR $FLAG[327] OR $FLAG[329]) AND ($IN[26] OR $IN[27]) AND $OUT[4039] THEN
            PREVSTEP = $APP_INT[5]
            $APP_INT[5] = 51
         ENDIF
      ;ENDFOLD
      ;FOLD Schritt 72 = (E785 & E804 & !E806 + E785 & E15 + F326 + F327 + F122) & A4039 ;%{SE}%MKUKATPVW %CVW_SPS %VST_CON %P 2:Schritt 72 = (E785 & E804 & !E806 + E785 & E15 + F326 + F327 + F122) & A4039, 3: ST_CON
         IF ($IN[785] AND $IN[804] AND NOT $IN[806] OR $IN[785] AND $IN[15] OR $FLAG[326] OR $FLAG[327] OR $FLAG[122]) AND $OUT[4039] THEN
            PREVSTEP = $APP_INT[5]
            $APP_INT[5] = 72
         ENDIF
      ;ENDFOLD
   ;ENDFOLD
   ;FOLD SCHRITT 72 -- STAT EZ1/SP1/KE1 -- ;%{P}%MKUKATPVW,%CSTEP,%VST_NR,%P 1:SCHRITT, 2:72, 3: STAT EZ1/SP1/KE1
      ;FOLD ;%{H}
         Case 72
      ;ENDFOLD
      ;FOLD A785 = AUS ;%{SE}%MKUKATPVW %CVW_SPS %VBOASG %P 2:A785 = AUS, 3: BOASG
         $OUT[785] = FALSE
      ;ENDFOLD
      ;FOLD F78 = !F327 & F78 ;%{SE}%MKUKATPVW %CVW_SPS %VBOASG %P 2:F78 = !F327 & F78, 3: BOASG
         $FLAG[78] = NOT $FLAG[327] AND $FLAG[78]
      ;ENDFOLD
      ;FOLD F79 = F327 + F79 ;%{SE}%MKUKATPVW %CVW_SPS %VBOASG %P 2:F79 = F327 + F79, 3: BOASG
         $FLAG[79] = $FLAG[327] OR $FLAG[79]
      ;ENDFOLD
      ;FOLD -- EZ1/SP1/KE1 SZ1 oeffnen -- ;%{SE}%MKUKATPVW %CVW_COM %VCOMMENT %P 2:-- EZ1/SP1/KE1 SZ1 oeffnen --, 3: VW_COMMENT
      ;ENDFOLD
      ;FOLD A718 = AUS ;%{SE}%MKUKATPVW %CVW_SPS %VBOASG %P 2:A718 = AUS, 3: BOASG
         $OUT[718] = FALSE
      ;ENDFOLD
      ;FOLD A766 = AUS ;%{SE}%MKUKATPVW %CVW_SPS %VBOASG %P 2:A766 = AUS, 3: BOASG
         $OUT[766] = FALSE
      ;ENDFOLD
      ;FOLD A717 = EIN ;%{SE}%MKUKATPVW %CVW_SPS %VBOASG %P 2:A717 = EIN, 3: BOASG
         $OUT[717] = TRUE
      ;ENDFOLD
      ;FOLD bin3 ( !F326 ) = 1 ;%{SE}%MKUKATPVW %CVW_SPS %VARIASG %P 2:bin3 ( !F326 ) = 1, 3: ARIASG
         VW(#BINOUT,NOT $FLAG[326],3,1)
      ;ENDFOLD
      ;FOLD -- Wartezeit Programmwechsel SK -- ;%{SE}%MKUKATPVW %CVW_COM %VCOMMENT %P 2:-- Wartezeit Programmwechsel SK --, 3: VW_COMMENT
      ;ENDFOLD
      ;FOLD T8 ( !F334 ) = -2[1/10Sek] ;%{SE}%MKUKATPVW %CVW_SPS %VTASG %P 2:T8 ( !F334 ) = -2[1/10Sek], 3: TASG
         VW(#SET_TIME,NOT $FLAG[334],8,0,-2)
      ;ENDFOLD
      ;FOLD -- Hilfsflag SK Programmwechsel -- ;%{SE}%MKUKATPVW %CVW_COM %VCOMMENT %P 2:-- Hilfsflag SK Programmwechsel --, 3: VW_COMMENT
      ;ENDFOLD
      ;FOLD F334 = EIN ;%{SE}%MKUKATPVW %CVW_SPS %VBOASG %P 2:F334 = EIN, 3: BOASG
         $FLAG[334] = TRUE
      ;ENDFOLD
      ;FOLD F748 = F322 + F323 + F325 + F326 + F327 + F329 ;%{SE}%MKUKATPVW %CVW_SPS %VBOASG %P 2:F748 = F322 + F323 + F325 + F326 + F327 + F329, 3: BOASG
         $FLAG[748] = $FLAG[322] OR $FLAG[323] OR $FLAG[325] OR $FLAG[326] OR $FLAG[327] OR $FLAG[329]
      ;ENDFOLD
      ;FOLD Schritt 51 = E717 & !E718 & (F322 + F323 + F325 + F326 + F327 + F329) & (E26 + E27) & A4039 ;%{SE}%MKUKATPVW %CVW_SPS %VST_CON %P 2:Schritt 51 = E717 & !E718 & (F322 + F323 + F325 + F326 + F327 + F329) & (E26 + E27) & A4039, 3: ST_CON
         IF $IN[717] AND NOT $IN[718] AND ($FLAG[322] OR $FLAG[323] OR $FLAG[325] OR $FLAG[326] OR $FLAG[327] OR $FLAG[329]) AND ($IN[26] OR $IN[27]) AND $OUT[4039] THEN
            PREVSTEP = $APP_INT[5]
            $APP_INT[5] = 51
         ENDIF
      ;ENDFOLD
      ;FOLD Schritt 51 = E717 & !E718 & (F322 + F323 + F325 + F326 + F327 + F329) & (F749 & F731) & A4039 ;%{SE}%MKUKATPVW %CVW_SPS %VST_CON %P 2:Schritt 51 = E717 & !E718 & (F322 + F323 + F325 + F326 + F327 + F329) & (F749 & F731) & A4039, 3: ST_CON
         IF $IN[717] AND NOT $IN[718] AND ($FLAG[322] OR $FLAG[323] OR $FLAG[325] OR $FLAG[326] OR $FLAG[327] OR $FLAG[329]) AND ($FLAG[749] AND $FLAG[731]) AND $OUT[4039] THEN
            PREVSTEP = $APP_INT[5]
            $APP_INT[5] = 51
         ENDIF
      ;ENDFOLD
      ;FOLD Schritt 73 = T8 & E717 & !E718 & (!F325 & !F326 & !F327 & !F329 + F122) & A4039 ;%{SE}%MKUKATPVW %CVW_SPS %VST_CON %P 2:Schritt 73 = T8 & E717 & !E718 & (!F325 & !F326 & !F327 & !F329 + F122) & A4039, 3: ST_CON
         IF $TIMER_FLAG[8] AND $IN[717] AND NOT $IN[718] AND (NOT $FLAG[325] AND NOT $FLAG[326] AND NOT $FLAG[327] AND NOT $FLAG[329] OR $FLAG[122]) AND $OUT[4039] THEN
            PREVSTEP = $APP_INT[5]
            $APP_INT[5] = 73
         ENDIF
      ;ENDFOLD
   ;ENDFOLD
   ;FOLD SCHRITT 73 -- STAT EZ1/SP1/KE1 # Ende -- ;%{P}%MKUKATPVW,%CSTEP,%VST_NR,%P 1:SCHRITT, 2:73, 3: STAT EZ1/SP1/KE1 # Ende
      ;FOLD ;%{H}
         Case 73
      ;ENDFOLD
      ;FOLD -- Hilfsflag SK Programmwechsel -- ;%{SE}%MKUKATPVW %CVW_COM %VCOMMENT %P 2:-- Hilfsflag SK Programmwechsel --, 3: VW_COMMENT
      ;ENDFOLD
      ;FOLD F334 = AUS ;%{SE}%MKUKATPVW %CVW_SPS %VBOASG %P 2:F334 = AUS, 3: BOASG
         $FLAG[334] = FALSE
      ;ENDFOLD
      ;FOLD -- RSK Sammelstoerung -- ;%{SE}%MKUKATPVW %CVW_COM %VCOMMENT %P 2:-- RSK Sammelstoerung --, 3: VW_COMMENT
      ;ENDFOLD
      ;FOLD F329 = F122 ;%{SE}%MKUKATPVW %CVW_SPS %VBOASG %P 2:F329 = F122, 3: BOASG
         $FLAG[329] = $FLAG[122]
      ;ENDFOLD
      ;FOLD F93 = !E786 & E787 & !E788 + F122 & (E26 + E27) ;%{SE}%MKUKATPVW %CVW_SPS %VBOASG %P 2:F93 = !E786 & E787 & !E788 + F122 & (E26 + E27), 3: BOASG
         $FLAG[93] = NOT $IN[786] AND $IN[787] AND NOT $IN[788] OR $FLAG[122] AND ($IN[26] OR $IN[27])
      ;ENDFOLD
      ;FOLD Schritt 1 = F93 & A4039 ;%{SE}%MKUKATPVW %CVW_SPS %VST_CON %P 2:Schritt 1 = F93 & A4039, 3: ST_CON
         IF $FLAG[93] AND $OUT[4039] THEN
            PREVSTEP = $APP_INT[5]
            $APP_INT[5] = 1
         ENDIF
      ;ENDFOLD
   ;ENDFOLD
   ;FOLD SCHRITT 74 -- STAT EZ2/SP2/KE2 # Start-- ;%{P}%MKUKATPVW,%CSTEP,%VST_NR,%P 1:SCHRITT, 2:74, 3: STAT EZ2/SP2/KE2 # Start
      ;FOLD ;%{H}
         Case 74
      ;ENDFOLD
      ;FOLD -- RSK gestartet -- ;%{SE}%MKUKATPVW %CVW_COM %VCOMMENT %P 2:-- RSK gestartet --, 3: VW_COMMENT
      ;ENDFOLD
      ;FOLD F160 = AUS ;%{SE}%MKUKATPVW %CVW_SPS %VBOASG %P 2:F160 = AUS, 3: BOASG
         $FLAG[160] = FALSE
      ;ENDFOLD
      ;FOLD F321 = AUS ;%{SE}%MKUKATPVW %CVW_SPS %VBOASG %P 2:F321 = AUS, 3: BOASG
         $FLAG[321] = FALSE
      ;ENDFOLD
      ;FOLD F322 = AUS ;%{SE}%MKUKATPVW %CVW_SPS %VBOASG %P 2:F322 = AUS, 3: BOASG
         $FLAG[322] = FALSE
      ;ENDFOLD
      ;FOLD F323 = AUS ;%{SE}%MKUKATPVW %CVW_SPS %VBOASG %P 2:F323 = AUS, 3: BOASG
         $FLAG[323] = FALSE
      ;ENDFOLD
      ;FOLD F324 = AUS ;%{SE}%MKUKATPVW %CVW_SPS %VBOASG %P 2:F324 = AUS, 3: BOASG
         $FLAG[324] = FALSE
      ;ENDFOLD
      ;FOLD F325 = AUS ;%{SE}%MKUKATPVW %CVW_SPS %VBOASG %P 2:F325 = AUS, 3: BOASG
         $FLAG[325] = FALSE
      ;ENDFOLD
      ;FOLD F326 = AUS ;%{SE}%MKUKATPVW %CVW_SPS %VBOASG %P 2:F326 = AUS, 3: BOASG
         $FLAG[326] = FALSE
      ;ENDFOLD
      ;FOLD F327 = AUS ;%{SE}%MKUKATPVW %CVW_SPS %VBOASG %P 2:F327 = AUS, 3: BOASG
         $FLAG[327] = FALSE
      ;ENDFOLD
      ;FOLD F329 = AUS ;%{SE}%MKUKATPVW %CVW_SPS %VBOASG %P 2:F329 = AUS, 3: BOASG
         $FLAG[329] = FALSE
      ;ENDFOLD
      ;FOLD -- EZ2/SP2/KE2 Zaehler -- ;%{SE}%MKUKATPVW %CVW_COM %VCOMMENT %P 2:-- EZ2/SP2/KE2 Zaehler --, 3: VW_COMMENT
      ;ENDFOLD
      ;FOLD F150 = AUS ;%{SE}%MKUKATPVW %CVW_SPS %VBOASG %P 2:F150 = AUS, 3: BOASG
         $FLAG[150] = FALSE
      ;ENDFOLD
      ;FOLD F151 = AUS ;%{SE}%MKUKATPVW %CVW_SPS %VBOASG %P 2:F151 = AUS, 3: BOASG
         $FLAG[151] = FALSE
      ;ENDFOLD
      ;FOLD F152 = AUS ;%{SE}%MKUKATPVW %CVW_SPS %VBOASG %P 2:F152 = AUS, 3: BOASG
         $FLAG[152] = FALSE
      ;ENDFOLD
      ;FOLD F153 = AUS ;%{SE}%MKUKATPVW %CVW_SPS %VBOASG %P 2:F153 = AUS, 3: BOASG
         $FLAG[153] = FALSE
      ;ENDFOLD
      ;FOLD F154 = AUS ;%{SE}%MKUKATPVW %CVW_SPS %VBOASG %P 2:F154 = AUS, 3: BOASG
         $FLAG[154] = FALSE
      ;ENDFOLD
      ;FOLD F155 = AUS ;%{SE}%MKUKATPVW %CVW_SPS %VBOASG %P 2:F155 = AUS, 3: BOASG
         $FLAG[155] = FALSE
      ;ENDFOLD
      ;FOLD -- Hilfsflags Funktionstest KF Motor -- ;%{SE}%MKUKATPVW %CVW_COM %VCOMMENT %P 2:-- Hilfsflags Funktionstest KF Motor --, 3: VW_COMMENT
      ;ENDFOLD
      ;FOLD F312 = AUS ;%{SE}%MKUKATPVW %CVW_SPS %VBOASG %P 2:F312 = AUS, 3: BOASG
         $FLAG[312] = FALSE
      ;ENDFOLD
      ;FOLD F313 = AUS ;%{SE}%MKUKATPVW %CVW_SPS %VBOASG %P 2:F313 = AUS, 3: BOASG
         $FLAG[313] = FALSE
      ;ENDFOLD
      ;FOLD bin3 ( F285 ) = 35 ;%{SE}%MKUKATPVW %CVW_SPS %VARIASG %P 2:bin3 ( F285 ) = 35, 3: ARIASG
         VW(#BINOUT,$FLAG[285],3,35)
      ;ENDFOLD
      ;FOLD bin4 ( !F831 ) = 31 ;%{SE}%MKUKATPVW %CVW_SPS %VARIASG %P 2:bin4 ( !F831 ) = 31, 3: ARIASG
         VW(#BINOUT,NOT $FLAG[831],4,31)
      ;ENDFOLD
      ;FOLD bin6 ( !F285 ) = 31 ;%{SE}%MKUKATPVW %CVW_SPS %VARIASG %P 2:bin6 ( !F285 ) = 31, 3: ARIASG
         VW(#BINOUT,NOT $FLAG[285],6,31)
      ;ENDFOLD
      ;FOLD -- Wartezeit Programmwechsel SK -- ;%{SE}%MKUKATPVW %CVW_COM %VCOMMENT %P 2:-- Wartezeit Programmwechsel SK --, 3: VW_COMMENT
      ;ENDFOLD
      ;FOLD T8 ( !F334 ) = -2[1/10Sek] ;%{SE}%MKUKATPVW %CVW_SPS %VTASG %P 2:T8 ( !F334 ) = -2[1/10Sek], 3: TASG
         VW(#SET_TIME,NOT $FLAG[334],8,0,-2)
      ;ENDFOLD
      ;FOLD -- Hilfsflag SK Programmwechsel -- ;%{SE}%MKUKATPVW %CVW_COM %VCOMMENT %P 2:-- Hilfsflag SK Programmwechsel --, 3: VW_COMMENT
      ;ENDFOLD
      ;FOLD F334 = EIN ;%{SE}%MKUKATPVW %CVW_SPS %VBOASG %P 2:F334 = EIN, 3: BOASG
         $FLAG[334] = TRUE
      ;ENDFOLD
      ;FOLD -- Quitt. Fraesen SK1 AUS -- ;%{SE}%MKUKATPVW %CVW_COM %VCOMMENT %P 2:-- Quitt. Fraesen SK1 AUS --, 3: VW_COMMENT
      ;ENDFOLD
      ;FOLD A786 = AUS ;%{SE}%MKUKATPVW %CVW_SPS %VBOASG %P 2:A786 = AUS, 3: BOASG
         $OUT[786] = FALSE
      ;ENDFOLD
      ;FOLD -- Quitt. Fraesen SK2 AUS -- ;%{SE}%MKUKATPVW %CVW_COM %VCOMMENT %P 2:-- Quitt. Fraesen SK2 AUS --, 3: VW_COMMENT
      ;ENDFOLD
      ;FOLD A946 = AUS ;%{SE}%MKUKATPVW %CVW_SPS %VBOASG %P 2:A946 = AUS, 3: BOASG
         $OUT[946] = FALSE
      ;ENDFOLD
      ;FOLD Schritt 75 = T8 & A4039 ;%{SE}%MKUKATPVW %CVW_SPS %VST_CON %P 2:Schritt 75 = T8 & A4039, 3: ST_CON
         IF $TIMER_FLAG[8] AND $OUT[4039] THEN
            PREVSTEP = $APP_INT[5]
            $APP_INT[5] = 75
         ENDIF
      ;ENDFOLD
   ;ENDFOLD
   ;FOLD SCHRITT 75 -- STAT EZ2/SP2/KE2 -- ;%{P}%MKUKATPVW,%CSTEP,%VST_NR,%P 1:SCHRITT, 2:75, 3: STAT EZ2/SP2/KE2
      ;FOLD ;%{H}
         Case 75
      ;ENDFOLD
      ;FOLD -- Fraeszyklen fuer autom. KF-Umderhung -- ;%{SE}%MKUKATPVW %CVW_COM %VCOMMENT %P 2:-- Fraeszyklen fuer autom. KF-Umderhung --, 3: VW_COMMENT
      ;ENDFOLD
      ;FOLD i36 (EIN) = i36 + 1 ;%{SE}%MKUKATPVW %CVW_SPS %VARIASG %P 2:i36 (EIN) = i36 + 1, 3: ARIASG
         VW(#COUNTER,TRUE,36,$COUNT_I[36] + 1)
      ;ENDFOLD
      ;FOLD -- Hilfsflag SK Programmwechsel -- ;%{SE}%MKUKATPVW %CVW_COM %VCOMMENT %P 2:-- Hilfsflag SK Programmwechsel --, 3: VW_COMMENT
      ;ENDFOLD
      ;FOLD F334 = AUS ;%{SE}%MKUKATPVW %CVW_SPS %VBOASG %P 2:F334 = AUS, 3: BOASG
         $FLAG[334] = FALSE
      ;ENDFOLD
      ;FOLD -- Ueberwachungszeit KF2 EIN -- ;%{SE}%MKUKATPVW %CVW_COM %VCOMMENT %P 2:-- Ueberwachungszeit KF2 EIN --, 3: VW_COMMENT
      ;ENDFOLD
      ;FOLD T7 ( EIN ) = -50[1/10Sek] ;%{SE}%MKUKATPVW %CVW_SPS %VTASG %P 2:T7 ( EIN ) = -50[1/10Sek], 3: TASG
         VW(#SET_TIME,TRUE,7,0,-50)
      ;ENDFOLD
      ;FOLD -- KF2 einschalten -- ;%{SE}%MKUKATPVW %CVW_COM %VCOMMENT %P 2:-- KF2 einschalten --, 3: VW_COMMENT
      ;ENDFOLD
      ;FOLD i1 (EIN) = 0 ;%{SE}%MKUKATPVW %CVW_SPS %VARIASG %P 2:i1 (EIN) = 0, 3: ARIASG
         VW(#COUNTER,TRUE,1,0)
      ;ENDFOLD
      ;FOLD A994 = EIN ;%{SE}%MKUKATPVW %CVW_SPS %VBOASG %P 2:A994 = EIN, 3: BOASG
         $OUT[994] = TRUE
      ;ENDFOLD
      ;FOLD Schritt 76 = A4039 ;%{SE}%MKUKATPVW %CVW_SPS %VST_CON %P 2:Schritt 76 = A4039, 3: ST_CON
         IF $OUT[4039] THEN
            PREVSTEP = $APP_INT[5]
            $APP_INT[5] = 76
         ENDIF
      ;ENDFOLD
   ;ENDFOLD
   ;FOLD SCHRITT 76 -- STAT EZ2/SP2/KE2 -- ;%{P}%MKUKATPVW,%CSTEP,%VST_NR,%P 1:SCHRITT, 2:76, 3: STAT EZ2/SP2/KE2
      ;FOLD ;%{H}
         Case 76
      ;ENDFOLD
      ;FOLD -- Funktionstest KF Motor -- ;%{SE}%MKUKATPVW %CVW_COM %VCOMMENT %P 2:-- Funktionstest KF Motor --, 3: VW_COMMENT
      ;ENDFOLD
      ;FOLD F312 = EIN ;%{SE}%MKUKATPVW %CVW_SPS %VBOASG %P 2:F312 = EIN, 3: BOASG
         $FLAG[312] = TRUE
      ;ENDFOLD
      ;FOLD F313 = i1 > 2 ;%{SE}%MKUKATPVW %CVW_SPS %VBOCMP %P 2:F313 = i1 > 2, 3: BOCMP
         $FLAG[313] = $COUNT_I[1] > 2
      ;ENDFOLD
      ;FOLD Schritt 77 = (F313 + T7) & A4039 ;%{SE}%MKUKATPVW %CVW_SPS %VST_CON %P 2:Schritt 77 = (F313 + T7) & A4039, 3: ST_CON
         IF ($FLAG[313] OR $TIMER_FLAG[7]) AND $OUT[4039] THEN
            PREVSTEP = $APP_INT[5]
            $APP_INT[5] = 77
         ENDIF
      ;ENDFOLD
   ;ENDFOLD
   ;FOLD SCHRITT 77 -- STAT EZ2/SP2/KE2-- ;%{P}%MKUKATPVW,%CSTEP,%VST_NR,%P 1:SCHRITT, 2:77, 3: STAT EZ2/SP2/KE2
      ;FOLD ;%{H}
         Case 77
      ;ENDFOLD
      ;FOLD F312 = AUS ;%{SE}%MKUKATPVW %CVW_SPS %VBOASG %P 2:F312 = AUS, 3: BOASG
         $FLAG[312] = FALSE
      ;ENDFOLD
      ;FOLD -- Ueberwachungszeit KS2 schwenken -- ;%{SE}%MKUKATPVW %CVW_COM %VCOMMENT %P 2:-- Ueberwachungszeit KS2 schwenken --, 3: VW_COMMENT
      ;ENDFOLD
      ;FOLD t8 ( EIN ) = -100[1/10Sek] ;%{SE}%MKUKATPVW %CVW_SPS %VTASG %P 2:t8 ( EIN ) = -100[1/10Sek], 3: TASG
         VW(#SET_TIME,TRUE,8,0,-100)
      ;ENDFOLD
      ;FOLD Schritt 78 = A4039 ;%{SE}%MKUKATPVW %CVW_SPS %VST_CON %P 2:Schritt 78 = A4039, 3: ST_CON
         IF $OUT[4039] THEN
            PREVSTEP = $APP_INT[5]
            $APP_INT[5] = 78
         ENDIF
      ;ENDFOLD
   ;ENDFOLD
   ;FOLD SCHRITT 78 -- STAT EZ2/SP2/KE2 -- ;%{P}%MKUKATPVW,%CSTEP,%VST_NR,%P 1:SCHRITT, 2:78, 3: STAT EZ2/SP2/KE2
      ;FOLD ;%{H}
         Case 78
      ;ENDFOLD
      ;FOLD -- RSK Fehlerausgabe KF1 Initiator/Motor -- ;%{SE}%MKUKATPVW %CVW_COM %VCOMMENT %P 2:-- RSK Fehlerausgabe KF1 Initiator/Motor --, 3: VW_COMMENT
      ;ENDFOLD
      ;FOLD F322 = !F313 ;%{SE}%MKUKATPVW %CVW_SPS %VBOASG %P 2:F322 = !F313, 3: BOASG
         $FLAG[322] = NOT $FLAG[313]
      ;ENDFOLD
      ;FOLD -- RSK Fehlerausgabe KS2 Ruhest. -- ;%{SE}%MKUKATPVW %CVW_COM %VCOMMENT %P 2:-- RSK Fehlerausgabe KS2 Ruhest. --, 3: VW_COMMENT
      ;ENDFOLD
      ;FOLD F323 = (!E996 + E997 + E998 + !E999) & !F324 & !F328 ;%{SE}%MKUKATPVW %CVW_SPS %VBOASG %P 2:F323 = (!E996 + E997 + E998 + !E999) & !F324 & !F328, 3: BOASG
         $FLAG[323] = (NOT $IN[996] OR $IN[997] OR $IN[998] OR NOT $IN[999]) AND NOT $FLAG[324] AND NOT $FLAG[328]
      ;ENDFOLD
      ;FOLD -- RSK Sammelstoerung -- ;%{SE}%MKUKATPVW %CVW_COM %VCOMMENT %P 2:-- RSK Sammelstoerung --, 3: VW_COMMENT
      ;ENDFOLD
      ;FOLD F329 = F322 + F323 ;%{SE}%MKUKATPVW %CVW_SPS %VBOASG %P 2:F329 = F322 + F323, 3: BOASG
         $FLAG[329] = $FLAG[322] OR $FLAG[323]
      ;ENDFOLD
      ;FOLD T7 ( EIN ) = STOP ;%{SE}%MKUKATPVW %CVW_SPS %VTSTOP %P 2:T7 ( EIN ) = STOP, 3: TSTOP
         VW(#SET_TIME,TRUE,7,1,0)
      ;ENDFOLD
      ;FOLD A994 = !F322 & !F323 ;%{SE}%MKUKATPVW %CVW_SPS %VBOASG %P 2:A994 = !F322 & !F323, 3: BOASG
         $OUT[994] = NOT $FLAG[322] AND NOT $FLAG[323]
      ;ENDFOLD
      ;FOLD -- KF2 Versetzeinheit vor -- ;%{SE}%MKUKATPVW %CVW_COM %VCOMMENT %P 2:-- KF2 Versetzeinheit vor --, 3: VW_COMMENT
      ;ENDFOLD
      ;FOLD A995 = !F322 & !F323 & F565 ;%{SE}%MKUKATPVW %CVW_SPS %VBOASG %P 2:A995 = !F322 & !F323 & F565, 3: BOASG
         $OUT[995] = NOT $FLAG[322] AND NOT $FLAG[323] AND $FLAG[565]
      ;ENDFOLD
      ;FOLD Schritt 79 = (!F322 & !F323 & (E995 & F565 + !E995 & !F565) + T8) & A4039 ;%{SE}%MKUKATPVW %CVW_SPS %VST_CON %P 2:Schritt 79 = (!F322 & !F323 & (E995 & F565 + !E995 & !F565) + T8) & A4039, 3: ST_CON
         IF (NOT $FLAG[322] AND NOT $FLAG[323] AND ($IN[995] AND $FLAG[565] OR NOT $IN[995] AND NOT $FLAG[565]) OR $TIMER_FLAG[8]) AND $OUT[4039] THEN
            PREVSTEP = $APP_INT[5]
            $APP_INT[5] = 79
         ENDIF
      ;ENDFOLD
      ;FOLD Schritt 95 = (F322 + F323) & !F324 & !F328 & A4039 ;%{SE}%MKUKATPVW %CVW_SPS %VST_CON %P 2:Schritt 95 = (F322 + F323) & !F324 & !F328 & A4039, 3: ST_CON
         IF ($FLAG[322] OR $FLAG[323]) AND NOT $FLAG[324] AND NOT $FLAG[328] AND $OUT[4039] THEN
            PREVSTEP = $APP_INT[5]
            $APP_INT[5] = 95
         ENDIF
      ;ENDFOLD
   ;ENDFOLD
   ;FOLD SCHRITT 79 -- STAT EZ2/SP2/KE2 -- ;%{P}%MKUKATPVW,%CSTEP,%VST_NR,%P 1:SCHRITT, 2:79, 3: STAT EZ2/SP2/KE2
      ;FOLD ;%{H}
         Case 79
      ;ENDFOLD
      ;FOLD -- RSK Sammelstoerung -- ;%{SE}%MKUKATPVW %CVW_COM %VCOMMENT %P 2:-- RSK Sammelstoerung --, 3: VW_COMMENT
      ;ENDFOLD
      ;FOLD F329 = T8 ;%{SE}%MKUKATPVW %CVW_SPS %VBOASG %P 2:F329 = T8, 3: BOASG
         $FLAG[329] = $TIMER_FLAG[8]
      ;ENDFOLD
      ;FOLD F324 = AUS ;%{SE}%MKUKATPVW %CVW_SPS %VBOASG %P 2:F324 = AUS, 3: BOASG
         $FLAG[324] = FALSE
      ;ENDFOLD
      ;FOLD F328 = AUS ;%{SE}%MKUKATPVW %CVW_SPS %VBOASG %P 2:F328 = AUS, 3: BOASG
         $FLAG[328] = FALSE
      ;ENDFOLD
      ;FOLD -- KS2 in Arbeitsstellung schwenken -- ;%{SE}%MKUKATPVW %CVW_COM %VCOMMENT %P 2:-- KS2 in Arbeitsstellung schwenken --, 3: VW_COMMENT
      ;ENDFOLD
      ;FOLD A1000 = (F746 + !F714) & E877 & !E997 & (E995 & F565 + !E995 & !F565) ;%{SE}%MKUKATPVW %CVW_SPS %VBOASG %P 2:A1000 = (F746 + !F714) & E877 & !E997 & (E995 & F565 + !E995 & !F565), 3: BOASG
         $OUT[1000] = ($FLAG[746] OR NOT $FLAG[714]) AND $IN[877] AND NOT $IN[997] AND ($IN[995] AND $FLAG[565] OR NOT $IN[995] AND NOT $FLAG[565])
      ;ENDFOLD
      ;FOLD -- KF2 Ausblasen -- ;%{SE}%MKUKATPVW %CVW_COM %VCOMMENT %P 2:-- KF2 Ausblasen --, 3: VW_COMMENT
      ;ENDFOLD
      ;FOLD A996 = F330 + !F330 & !F331 & !F332 ;%{SE}%MKUKATPVW %CVW_SPS %VBOASG %P 2:A996 = F330 + !F330 & !F331 & !F332, 3: BOASG
         $OUT[996] = $FLAG[330] OR NOT $FLAG[330] AND NOT $FLAG[331] AND NOT $FLAG[332]
      ;ENDFOLD
      ;FOLD Schritt 80 = (F746 + !F714) & E877 & (A1000 + E997 + T8) & A4039 ;%{SE}%MKUKATPVW %CVW_SPS %VST_CON %P 2:Schritt 80 = (F746 + !F714) & E877 & (A1000 + E997 + T8) & A4039, 3: ST_CON
         IF ($FLAG[746] OR NOT $FLAG[714]) AND $IN[877] AND ($OUT[1000] OR $IN[997] OR $TIMER_FLAG[8]) AND $OUT[4039] THEN
            PREVSTEP = $APP_INT[5]
            $APP_INT[5] = 80
         ENDIF
      ;ENDFOLD
   ;ENDFOLD
   ;FOLD SCHRITT 80 -- STAT EZ2/SP2/KE2 -- ;%{P}%MKUKATPVW,%CSTEP,%VST_NR,%P 1:SCHRITT, 2:80, 3: STAT EZ2/SP2/KE2
      ;FOLD ;%{H}
         Case 80
      ;ENDFOLD
      ;FOLD -- RSK Fehlerausgabe KF Versetzeinheit -- ;%{SE}%MKUKATPVW %CVW_COM %VCOMMENT %P 2:-- RSK Fehlerausgabe KF Versetzeinheit --, 3: VW_COMMENT
      ;ENDFOLD
      ;FOLD F328 = !E995 & F565 & !F324 ;%{SE}%MKUKATPVW %CVW_SPS %VBOASG %P 2:F328 = !E995 & F565 & !F324, 3: BOASG
         $FLAG[328] = NOT $IN[995] AND $FLAG[565] AND NOT $FLAG[324]
      ;ENDFOLD
      ;FOLD -- RSK Fehlerausgabe KS2 Arbeitsstellung -- ;%{SE}%MKUKATPVW %CVW_COM %VCOMMENT %P 2:-- RSK Fehlerausgabe KS2 Arbeitsstellung --, 3: VW_COMMENT
      ;ENDFOLD
      ;FOLD F324 = (E996 + !E997 + !E998 + E999) & T8 & (E995 + !F565) + F324 ;%{SE}%MKUKATPVW %CVW_SPS %VBOASG %P 2:F324 = (E996 + !E997 + !E998 + E999) & T8 & (E995 + !F565) + F324, 3: BOASG
         $FLAG[324] = ($IN[996] OR NOT $IN[997] OR NOT $IN[998] OR $IN[999]) AND $TIMER_FLAG[8] AND ($IN[995] OR NOT $FLAG[565]) OR $FLAG[324]
      ;ENDFOLD
      ;FOLD -- RSK Fehlerausgabe EZ/SP min. Oeffnung -- ;%{SE}%MKUKATPVW %CVW_COM %VCOMMENT %P 2:-- RSK Fehlerausgabe EZ/SP min. Oeffnung --, 3: VW_COMMENT
      ;ENDFOLD
      ;FOLD F333 = !F746 ;%{SE}%MKUKATPVW %CVW_SPS %VBOASG %P 2:F333 = !F746, 3: BOASG
         $FLAG[333] = NOT $FLAG[746]
      ;ENDFOLD
      ;FOLD -- RSK Sammelstoerung -- ;%{SE}%MKUKATPVW %CVW_COM %VCOMMENT %P 2:-- RSK Sammelstoerung --, 3: VW_COMMENT
      ;ENDFOLD
      ;FOLD F329 = F324 + F328 + F333 ;%{SE}%MKUKATPVW %CVW_SPS %VBOASG %P 2:F329 = F324 + F328 + F333, 3: BOASG
         $FLAG[329] = $FLAG[324] OR $FLAG[328] OR $FLAG[333]
      ;ENDFOLD
      ;FOLD A994 = !F324 & !F328 ;%{SE}%MKUKATPVW %CVW_SPS %VBOASG %P 2:A994 = !F324 & !F328, 3: BOASG
         $OUT[994] = NOT $FLAG[324] AND NOT $FLAG[328]
      ;ENDFOLD
      ;FOLD -- KF1 Ausblasen -- ;%{SE}%MKUKATPVW %CVW_COM %VCOMMENT %P 2:-- KF1 Ausblasen --, 3: VW_COMMENT
      ;ENDFOLD
      ;FOLD A996 = (F330 + !F330 & !F331 & !F332) & !F324 & !F328 ;%{SE}%MKUKATPVW %CVW_SPS %VBOASG %P 2:A996 = (F330 + !F330 & !F331 & !F332) & !F324 & !F328, 3: BOASG
         $OUT[996] = ($FLAG[330] OR NOT $FLAG[330] AND NOT $FLAG[331] AND NOT $FLAG[332]) AND NOT $FLAG[324] AND NOT $FLAG[328]
      ;ENDFOLD
      ;FOLD A995 = F565 ;%{SE}%MKUKATPVW %CVW_SPS %VBOASG %P 2:A995 = F565, 3: BOASG
         $OUT[995] = $FLAG[565]
      ;ENDFOLD
      ;FOLD -- Ueberwachungszeit EZ2/SP2/KE2 schliessen -- ;%{SE}%MKUKATPVW %CVW_COM %VCOMMENT %P 2:-- Ueberwachungszeit EZ2/SP2/KE2 schliessen --, 3: VW_COMMENT
      ;ENDFOLD
      ;FOLD t9 ( EIN ) = -80[1/10Sek] ;%{SE}%MKUKATPVW %CVW_SPS %VTASG %P 2:t9 ( EIN ) = -80[1/10Sek], 3: TASG
         VW(#SET_TIME,TRUE,9,0,-80)
      ;ENDFOLD
      ;FOLD -- Verweilzeit Versetzeinheit Rueck -- ;%{SE}%MKUKATPVW %CVW_COM %VCOMMENT %P 2:-- Verweilzeit Versetzeinheit Rueck --, 3: VW_COMMENT
      ;ENDFOLD
      ;FOLD t11 ( EIN ) = i24[1/10Sek] ;%{SE}%MKUKATPVW %CVW_SPS %VTASG %P 2:t11 ( EIN ) = i24[1/10Sek], 3: TASG
         VW(#SET_TIME,TRUE,11,0,$COUNT_I[24])
      ;ENDFOLD
      ;FOLD Schritt 75 = (F324 + F328) & (E26 + E27) & A4039 ;%{SE}%MKUKATPVW %CVW_SPS %VST_CON %P 2:Schritt 75 = (F324 + F328) & (E26 + E27) & A4039, 3: ST_CON
         IF ($FLAG[324] OR $FLAG[328]) AND ($IN[26] OR $IN[27]) AND $OUT[4039] THEN
            PREVSTEP = $APP_INT[5]
            $APP_INT[5] = 75
         ENDIF
      ;ENDFOLD
      ;FOLD Schritt 81 = !F324 & !F328 & !E996 & E997 & E998 & !E999 & A4039 ;%{SE}%MKUKATPVW %CVW_SPS %VST_CON %P 2:Schritt 81 = !F324 & !F328 & !E996 & E997 & E998 & !E999 & A4039, 3: ST_CON
         IF NOT $FLAG[324] AND NOT $FLAG[328] AND NOT $IN[996] AND $IN[997] AND $IN[998] AND NOT $IN[999] AND $OUT[4039] THEN
            PREVSTEP = $APP_INT[5]
            $APP_INT[5] = 81
         ENDIF
      ;ENDFOLD
   ;ENDFOLD
   ;FOLD SCHRITT 81 -- STAT EZ2/SP2/KE2-- ;%{P}%MKUKATPVW,%CSTEP,%VST_NR,%P 1:SCHRITT, 2:81, 3: STAT EZ2/SP2/KE2
      ;FOLD ;%{H}
         Case 81
      ;ENDFOLD
      ;FOLD -- Umdreh. KF setzen zwischenspeichern -- ;%{SE}%MKUKATPVW %CVW_COM %VCOMMENT %P 2:-- Umdreh. KF setzen zwischenspeichern --, 3: VW_COMMENT
      ;ENDFOLD
      ;FOLD i45 ( EIN ) = i7 ;%{SE}%MKUKATPVW %CVW_SPS %VARIASG %P 2:i45 ( EIN ) = i7, 3: ARIASG
         VW(#COUNTER,TRUE,45,$COUNT_I[7])
      ;ENDFOLD
      ;FOLD i4 ( F155 ) = i43 ;%{SE}%MKUKATPVW %CVW_SPS %VARIASG %P 2:i4 ( F155 ) = i43, 3: ARIASG
         VW(#COUNTER,$FLAG[155],4,$COUNT_I[43])
      ;ENDFOLD
      ;FOLD i1 ( EIN ) = 0 ;%{SE}%MKUKATPVW %CVW_SPS %VARIASG %P 2:i1 ( EIN ) = 0, 3: ARIASG
         VW(#COUNTER,TRUE,1,0)
      ;ENDFOLD
      ;FOLD F154 = AUS ;%{SE}%MKUKATPVW %CVW_SPS %VBOASG %P 2:F154 = AUS, 3: BOASG
         $FLAG[154] = FALSE
      ;ENDFOLD
      ;FOLD F312 = AUS ;%{SE}%MKUKATPVW %CVW_SPS %VBOASG %P 2:F312 = AUS, 3: BOASG
         $FLAG[312] = FALSE
      ;ENDFOLD
      ;FOLD F313 = AUS ;%{SE}%MKUKATPVW %CVW_SPS %VBOASG %P 2:F313 = AUS, 3: BOASG
         $FLAG[313] = FALSE
      ;ENDFOLD
      ;FOLD F324 = AUS ;%{SE}%MKUKATPVW %CVW_SPS %VBOASG %P 2:F324 = AUS, 3: BOASG
         $FLAG[324] = FALSE
      ;ENDFOLD
      ;FOLD F328 = AUS ;%{SE}%MKUKATPVW %CVW_SPS %VBOASG %P 2:F328 = AUS, 3: BOASG
         $FLAG[328] = FALSE
      ;ENDFOLD
      ;FOLD -- KF2 einschalten nach Fehler -- ;%{SE}%MKUKATPVW %CVW_COM %VCOMMENT %P 2:-- KF2 einschalten nach Fehler --, 3: VW_COMMENT
      ;ENDFOLD
      ;FOLD A994 = EIN ;%{SE}%MKUKATPVW %CVW_SPS %VBOASG %P 2:A994 = EIN, 3: BOASG
         $OUT[994] = TRUE
      ;ENDFOLD
      ;FOLD -- KF2 Versetzeinheit rueck -- ;%{SE}%MKUKATPVW %CVW_COM %VCOMMENT %P 2:-- KF2 Versetzeinheit rueck --, 3: VW_COMMENT
      ;ENDFOLD
      ;FOLD A995 = AUS ;%{SE}%MKUKATPVW %CVW_SPS %VBOASG %P 2:A995 = AUS, 3: BOASG
         $OUT[995] = FALSE
      ;ENDFOLD
      ;FOLD Schritt 82 = T11 & A4039 ;%{SE}%MKUKATPVW %CVW_SPS %VST_CON %P 2:Schritt 82 = T11 & A4039, 3: ST_CON
         IF $TIMER_FLAG[11] AND $OUT[4039] THEN
            PREVSTEP = $APP_INT[5]
            $APP_INT[5] = 82
         ENDIF
      ;ENDFOLD
   ;ENDFOLD
   ;FOLD SCHRITT 82 -- STAT EZ2/SP2/KE2 -- ;%{P}%MKUKATPVW,%CSTEP,%VST_NR,%P 1:SCHRITT, 2:82, 3: STAT EZ2/SP2/KE2
      ;FOLD ;%{H}
         Case 82
      ;ENDFOLD
      ;FOLD t11 ( EIN ) = STOP ;%{SE}%MKUKATPVW %CVW_SPS %VTSTOP %P 2:t11 ( EIN ) = STOP, 3: TSTOP
         VW(#SET_TIME,TRUE,11,1,0)
      ;ENDFOLD
      ;FOLD -- EZ2/SP2/KE2 schliessen -- ;%{SE}%MKUKATPVW %CVW_COM %VCOMMENT %P 2:-- EZ2/SP2/KE2 schliessen --, 3: VW_COMMENT
      ;ENDFOLD
      ;FOLD A877 = AUS ;%{SE}%MKUKATPVW %CVW_SPS %VBOASG %P 2:A877 = AUS, 3: BOASG
         $OUT[877] = FALSE
      ;ENDFOLD
      ;FOLD -- EZ2/SP2 -- ;%{SE}%MKUKATPVW %CVW_COM %VCOMMENT %P 2:-- EZ2/SP2 --, 3: VW_COMMENT
      ;ENDFOLD
      ;FOLD A878 = !F831 ;%{SE}%MKUKATPVW %CVW_SPS %VBOASG %P 2:A878 = !F831, 3: BOASG
         $OUT[878] = NOT $FLAG[831]
      ;ENDFOLD
      ;FOLD -- KE2 -- ;%{SE}%MKUKATPVW %CVW_COM %VCOMMENT %P 2:-- KE2 --, 3: VW_COMMENT
      ;ENDFOLD
      ;FOLD A926 = F831 ;%{SE}%MKUKATPVW %CVW_SPS %VBOASG %P 2:A926 = F831, 3: BOASG
         $OUT[926] = $FLAG[831]
      ;ENDFOLD
      ;FOLD -- KF2 Ausblasen -- ;%{SE}%MKUKATPVW %CVW_COM %VCOMMENT %P 2:-- KF2 Ausblasen --, 3: VW_COMMENT
      ;ENDFOLD
      ;FOLD A996 = F330 + F331 + !F330 & !F331 & !F332 ;%{SE}%MKUKATPVW %CVW_SPS %VBOASG %P 2:A996 = F330 + F331 + !F330 & !F331 & !F332, 3: BOASG
         $OUT[996] = $FLAG[330] OR $FLAG[331] OR NOT $FLAG[330] AND NOT $FLAG[331] AND NOT $FLAG[332]
      ;ENDFOLD
      ;FOLD Schritt 83 = (!E877 & E878 + T9) & A4039 ;%{SE}%MKUKATPVW %CVW_SPS %VST_CON %P 2:Schritt 83 = (!E877 & E878 + T9) & A4039, 3: ST_CON
         IF (NOT $IN[877] AND $IN[878] OR $TIMER_FLAG[9]) AND $OUT[4039] THEN
            PREVSTEP = $APP_INT[5]
            $APP_INT[5] = 83
         ENDIF
      ;ENDFOLD
   ;ENDFOLD
   ;FOLD SCHRITT 83 -- STAT EZ2/SP2/KE2 -- ;%{P}%MKUKATPVW,%CSTEP,%VST_NR,%P 1:SCHRITT, 2:83, 3: STAT EZ2/SP2/KE2
      ;FOLD ;%{H}
         Case 83
      ;ENDFOLD
      ;FOLD -- RSK Fehlerausgabe Kraftaufbau -- ;%{SE}%MKUKATPVW %CVW_COM %VCOMMENT %P 2:-- RSK Fehlerausgabe Kraftaufbau --, 3: VW_COMMENT
      ;ENDFOLD
      ;FOLD F325 = T9 ;%{SE}%MKUKATPVW %CVW_SPS %VBOASG %P 2:F325 = T9, 3: BOASG
         $FLAG[325] = $TIMER_FLAG[9]
      ;ENDFOLD
      ;FOLD -- RSK Sammelstoerung -- ;%{SE}%MKUKATPVW %CVW_COM %VCOMMENT %P 2:-- RSK Sammelstoerung --, 3: VW_COMMENT
      ;ENDFOLD
      ;FOLD F329 = F325 ;%{SE}%MKUKATPVW %CVW_SPS %VBOASG %P 2:F329 = F325, 3: BOASG
         $FLAG[329] = $FLAG[325]
      ;ENDFOLD
      ;FOLD -- KF2 abschalten bei Fehler -- ;%{SE}%MKUKATPVW %CVW_COM %VCOMMENT %P 2:-- KF2 abschalten bei Fehler --, 3: VW_COMMENT
      ;ENDFOLD
      ;FOLD A994 = !T9 ;%{SE}%MKUKATPVW %CVW_SPS %VBOASG %P 2:A994 = !T9, 3: BOASG
         $OUT[994] = NOT $TIMER_FLAG[9]
      ;ENDFOLD
      ;FOLD -- KF2 Ausblasen -- ;%{SE}%MKUKATPVW %CVW_COM %VCOMMENT %P 2:-- KF2 Ausblasen --, 3: VW_COMMENT
      ;ENDFOLD
      ;FOLD A996 = (F330 + F331 + !F330 & !F331 & !F332) & !T9 ;%{SE}%MKUKATPVW %CVW_SPS %VBOASG %P 2:A996 = (F330 + F331 + !F330 & !F331 & !F332) & !T9, 3: BOASG
         $OUT[996] = ($FLAG[330] OR $FLAG[331] OR NOT $FLAG[330] AND NOT $FLAG[331] AND NOT $FLAG[332]) AND NOT $TIMER_FLAG[9]
      ;ENDFOLD
      ;FOLD -- Warte Fraesen fertig oder Timeout -- ;%{SE}%MKUKATPVW %CVW_COM %VCOMMENT %P 2:-- Warte Fraesen fertig oder Timeout --, 3: VW_COMMENT
      ;ENDFOLD
      ;FOLD Schritt 84 = (F139 & F154 + F138 & F150 & !F287 + T7 + T9 + F325) & A4039 ;%{SE}%MKUKATPVW %CVW_SPS %VST_CON %P 2:Schritt 84 = (F139 & F154 + F138 & F150 & !F287 + T7 + T9 + F325) & A4039, 3: ST_CON
         IF ($FLAG[139] AND $FLAG[154] OR $FLAG[138] AND $FLAG[150] AND NOT $FLAG[287] OR $TIMER_FLAG[7] OR $TIMER_FLAG[9] OR $FLAG[325]) AND $OUT[4039] THEN
            PREVSTEP = $APP_INT[5]
            $APP_INT[5] = 84
         ENDIF
      ;ENDFOLD
      ;FOLD Schritt 84 = (F138 & F152 & F287 + T7 + T9 + F325) & A4039 ;%{SE}%MKUKATPVW %CVW_SPS %VST_CON %P 2:Schritt 84 = (F138 & F152 & F287 + T7 + T9 + F325) & A4039, 3: ST_CON
         IF ($FLAG[138] AND $FLAG[152] AND $FLAG[287] OR $TIMER_FLAG[7] OR $TIMER_FLAG[9] OR $FLAG[325]) AND $OUT[4039] THEN
            PREVSTEP = $APP_INT[5]
            $APP_INT[5] = 84
         ENDIF
      ;ENDFOLD
   ;ENDFOLD
   ;FOLD SCHRITT 84 -- STAT EZ2/SP2/KE2-- ;%{P}%MKUKATPVW,%CSTEP,%VST_NR,%P 1:SCHRITT, 2:84, 3: STAT EZ2/SP2/KE2
      ;FOLD ;%{H}
         Case 84
      ;ENDFOLD
      ;FOLD t9 ( EIN ) = STOP ;%{SE}%MKUKATPVW %CVW_SPS %VTSTOP %P 2:t9 ( EIN ) = STOP, 3: TSTOP
         VW(#SET_TIME,TRUE,9,1,0)
      ;ENDFOLD
      ;FOLD -- EZ2/SP2/KE2 oeffnen -- ;%{SE}%MKUKATPVW %CVW_COM %VCOMMENT %P 2:-- EZ2/SP2/KE2 oeffnen --, 3: VW_COMMENT
      ;ENDFOLD
      ;FOLD A878 = AUS ;%{SE}%MKUKATPVW %CVW_SPS %VBOASG %P 2:A878 = AUS, 3: BOASG
         $OUT[878] = FALSE
      ;ENDFOLD
      ;FOLD A926 = AUS ;%{SE}%MKUKATPVW %CVW_SPS %VBOASG %P 2:A926 = AUS, 3: BOASG
         $OUT[926] = FALSE
      ;ENDFOLD
      ;FOLD A877 = EIN ;%{SE}%MKUKATPVW %CVW_SPS %VBOASG %P 2:A877 = EIN, 3: BOASG
         $OUT[877] = TRUE
      ;ENDFOLD
      ;FOLD -- KF2 Ausblasen -- ;%{SE}%MKUKATPVW %CVW_COM %VCOMMENT %P 2:-- KF2 Ausblasen --, 3: VW_COMMENT
      ;ENDFOLD
      ;FOLD A996 = F330 + F331 + F332 + !F330 & !F331 & !F332 ;%{SE}%MKUKATPVW %CVW_SPS %VBOASG %P 2:A996 = F330 + F331 + F332 + !F330 & !F331 & !F332, 3: BOASG
         $OUT[996] = $FLAG[330] OR $FLAG[331] OR $FLAG[332] OR NOT $FLAG[330] AND NOT $FLAG[331] AND NOT $FLAG[332]
      ;ENDFOLD
      ;FOLD -- KF Ausblasen Ausschaltverzoegerung starten -- ;%{SE}%MKUKATPVW %CVW_COM %VCOMMENT %P 2:-- KF Ausblasen Ausschaltverzoegerung starten --, 3: VW_COMMENT
      ;ENDFOLD
      ;FOLD F738 = EIN ;%{SE}%MKUKATPVW %CVW_SPS %VBOASG %P 2:F738 = EIN, 3: BOASG
         $FLAG[738] = TRUE
      ;ENDFOLD
